LIN {X 0,Y 488.244,Z 843.404,A -85,B 0,C 180,E1 -6577.215,E2 -6577.215} C_VEL
LIN {X 0,Y 488.428,Z 836.225,A -85,B 0,C 180,E1 -6578.482,E2 -6578.482} C_VEL
LIN {X 0,Y 488.619,Z 827.431,A -85,B 0,C 180,E1 -6579.73,E2 -6579.73} C_VEL
LIN {X 0,Y 488.934,Z 817.433,A -85,B 0,C 180,E1 -6580.875,E2 -6580.875} C_VEL
LIN {X 0,Y 489.324,Z 806.303,A -85,B 0,C 180,E1 -6581.902,E2 -6581.902} C_VEL
LIN {X 0,Y 489.653,Z 795.065,A -85,B 0,C 180,E1 -6582.738,E2 -6582.738} C_VEL
LIN {X 0,Y 490.023,Z 782.384,A -85,B 0,C 180,E1 -6583.478,E2 -6583.478} C_VEL
LIN {X 0,Y 490.49,Z 769.48,A -85,B 0,C 180,E1 -6584.046,E2 -6584.046} C_VEL
LIN {X 0,Y 490.805,Z 756.071,A -85,B 0,C 180,E1 -6584.46,E2 -6584.46} C_VEL
LIN {X 0,Y 491.062,Z 737.319,A -85,B 0,C 180,E1 -6584.796,E2 -6584.796} C_VEL
LIN {X 0,Y 491.554,Z 664.239,A -85,B 0,C 180,E1 -6585.948,E2 -6585.948} C_VEL
LIN {X 0,Y 490.064,Z 652.447,A -85,B 0,C 180,E1 -6586.19,E2 -6586.19} C_VEL
LIN {X 0,Y 489.098,Z 638.268,A -85,B 0,C 180,E1 -6586.485,E2 -6586.485} C_VEL
LIN {X 0,Y 489.362,Z 617.504,A -85,B 0,C 180,E1 -6589.506,E2 -6589.506} C_VEL
LIN {X 0,Y 489.557,Z 597.975,A -85,B 0,C 180,E1 -6592.361,E2 -6592.361} C_VEL
LIN {X 0,Y 489.714,Z 578.159,A -85,B 0,C 180,E1 -6595.293,E2 -6595.293} C_VEL
LIN {X 0,Y 489.897,Z 557.152,A -85,B 0,C 180,E1 -6598.468,E2 -6598.468} C_VEL
LIN {X 0,Y 489.78,Z 545.178,A -85,B 0,C 180,E1 -6600.327,E2 -6600.327} C_VEL
LIN {X 0,Y 488.831,Z 539.598,A -85,B 0,C 180,E1 -6601.261,E2 -6601.261} C_VEL
LIN {X 0,Y 488.737,Z 539.605,A -85,B 0,C 180,E1 -6604.113,E2 -6604.113} C_VEL
LIN {X 0,Y 488.684,Z 539.613,A -85,B 0,C 180,E1 -6607.159,E2 -6607.159} C_VEL
LIN {X 0,Y 488.723,Z 539.606,A -85,B 0,C 180,E1 -6610.345,E2 -6610.345} C_VEL
LIN {X 0,Y 488.691,Z 539.608,A -85,B 0,C 180,E1 -6613.654,E2 -6613.654} C_VEL
LIN {X 0,Y 488.692,Z 539.611,A -85,B 0,C 180,E1 -6616.346,E2 -6616.346} C_VEL
LIN {X 0,Y 488.737,Z 539.602,A -85,B 0,C 180,E1 -6619.677,E2 -6619.677} C_VEL
LIN {X 0,Y 488.684,Z 539.615,A -85,B 0,C 180,E1 -6622.841,E2 -6622.841} C_VEL
LIN {X 0,Y 488.735,Z 539.604,A -85,B 0,C 180,E1 -6625.887,E2 -6625.887} C_VEL
LIN {X 0,Y 488.697,Z 539.612,A -85,B 0,C 180,E1 -6628.82,E2 -6628.82} C_VEL
LIN {X 0,Y 488.75,Z 539.602,A -85,B 0,C 180,E1 -6631.671,E2 -6631.671} C_VEL
LIN {X 0,Y 488.752,Z 539.608,A -85,B 0,C 180,E1 -6634.444,E2 -6634.444} C_VEL
LIN {X 0,Y 488.728,Z 539.607,A -85,B 0,C 180,E1 -6637.153,E2 -6637.153} C_VEL
LIN {X 0,Y 488.73,Z 539.607,A -85,B 0,C 180,E1 -6639.81,E2 -6639.81} C_VEL
LIN {X 0,Y 488.751,Z 539.609,A -85,B 0,C 180,E1 -6642.591,E2 -6642.591} C_VEL
LIN {X 0,Y 492.762,Z 551.195,A -85,B 0,C 180,E1 -6642.917,E2 -6642.917} C_VEL
LIN {X 0,Y 492.751,Z 584.57,A -85,B 0,C 180,E1 -6643.426,E2 -6643.426} C_VEL
LIN {X 0,Y 492.704,Z 599.838,A -85,B 0,C 180,E1 -6643.83,E2 -6643.83} C_VEL
LIN {X 0,Y 492.57,Z 614.087,A -85,B 0,C 180,E1 -6644.377,E2 -6644.377} C_VEL
LIN {X 0,Y 492.273,Z 626.69,A -85,B 0,C 180,E1 -6645.003,E2 -6645.003} C_VEL
LIN {X 0,Y 491.859,Z 639.98,A -85,B 0,C 180,E1 -6645.836,E2 -6645.836} C_VEL
LIN {X 0,Y 491.447,Z 653.278,A -85,B 0,C 180,E1 -6646.878,E2 -6646.878} C_VEL
LIN {X 0,Y 491.009,Z 664.22,A -85,B 0,C 180,E1 -6647.916,E2 -6647.916} C_VEL
LIN {X 0,Y 490.483,Z 674.33,A -85,B 0,C 180,E1 -6649.055,E2 -6649.055} C_VEL
LIN {X 0,Y 489.999,Z 683.621,A -85,B 0,C 180,E1 -6650.297,E2 -6650.297} C_VEL
LIN {X 0,Y 489.615,Z 692.638,A -85,B 0,C 180,E1 -6651.747,E2 -6651.747} C_VEL
LIN {X 0,Y 489.34,Z 699.094,A -85,B 0,C 180,E1 -6652.988,E2 -6652.988} C_VEL
LIN {X 0,Y 488.977,Z 704.583,A -85,B 0,C 180,E1 -6654.225,E2 -6654.225} C_VEL
LIN {X 0,Y 488.744,Z 710.483,A -85,B 0,C 180,E1 -6655.877,E2 -6655.877} C_VEL
LIN {X 0,Y 488.548,Z 714.977,A -85,B 0,C 180,E1 -6657.526,E2 -6657.526} C_VEL
LIN {X 0,Y 488.433,Z 718.193,A -85,B 0,C 180,E1 -6659.175,E2 -6659.175} C_VEL
LIN {X 0,Y 488.414,Z 720.216,A -85,B 0,C 180,E1 -6660.824,E2 -6660.824} C_VEL
LIN {X 0,Y 488.451,Z 721.099,A -85,B 0,C 180,E1 -6662.474,E2 -6662.474} C_VEL
LIN {X 0,Y 488.351,Z 720.88,A -85,B 0,C 180,E1 -6664.126,E2 -6664.126} C_VEL
LIN {X 0,Y 488.426,Z 719.509,A -85,B 0,C 180,E1 -6665.78,E2 -6665.78} C_VEL
LIN {X 0,Y 488.492,Z 716.945,A -85,B 0,C 180,E1 -6667.439,E2 -6667.439} C_VEL
LIN {X 0,Y 488.66,Z 713.137,A -85,B 0,C 180,E1 -6669.102,E2 -6669.102} C_VEL
LIN {X 0,Y 488.734,Z 708.023,A -85,B 0,C 180,E1 -6670.774,E2 -6670.774} C_VEL
LIN {X 0,Y 489.054,Z 701.415,A -85,B 0,C 180,E1 -6672.448,E2 -6672.448} C_VEL
LIN {X 0,Y 489.458,Z 693.105,A -85,B 0,C 180,E1 -6674.128,E2 -6674.128} C_VEL
LIN {X 0,Y 489.883,Z 684.147,A -85,B 0,C 180,E1 -6675.604,E2 -6675.604} C_VEL
LIN {X 0,Y 490.418,Z 673.246,A -85,B 0,C 180,E1 -6677.084,E2 -6677.084} C_VEL
LIN {X 0,Y 490.971,Z 661.901,A -85,B 0,C 180,E1 -6678.355,E2 -6678.355} C_VEL
LIN {X 0,Y 491.484,Z 650.595,A -85,B 0,C 180,E1 -6679.418,E2 -6679.418} C_VEL
LIN {X 0,Y 491.957,Z 638.327,A -85,B 0,C 180,E1 -6680.378,E2 -6680.378} C_VEL
LIN {X 0,Y 492.432,Z 624.976,A -85,B 0,C 180,E1 -6681.232,E2 -6681.232} C_VEL
LIN {X 0,Y 492.849,Z 612.015,A -85,B 0,C 180,E1 -6681.893,E2 -6681.893} C_VEL
LIN {X 0,Y 493.158,Z 597.332,A -85,B 0,C 180,E1 -6682.474,E2 -6682.474} C_VEL
LIN {X 0,Y 493.277,Z 584.102,A -85,B 0,C 180,E1 -6682.855,E2 -6682.855} C_VEL
LIN {X 0,Y 493.378,Z 564.328,A -85,B 0,C 180,E1 -6683.214,E2 -6683.214} C_VEL
LIN {X 0,Y 493.335,Z 552.237,A -85,B 0,C 180,E1 -6683.406,E2 -6683.406} C_VEL
LIN {X 0,Y 488.739,Z 539.609,A -85,B 0,C 180,E1 -6683.799,E2 -6683.799} C_VEL
LIN {X 0,Y 488.794,Z 539.595,A -85,B 0,C 180,E1 -6686.943,E2 -6686.943} C_VEL
LIN {X 0,Y 488.711,Z 539.608,A -85,B 0,C 180,E1 -6690.362,E2 -6690.362} C_VEL
LIN {X 0,Y 488.735,Z 539.602,A -85,B 0,C 180,E1 -6693.484,E2 -6693.484} C_VEL
LIN {X 0,Y 488.683,Z 539.613,A -85,B 0,C 180,E1 -6696.354,E2 -6696.354} C_VEL
LIN {X 0,Y 488.703,Z 539.604,A -85,B 0,C 180,E1 -6699.254,E2 -6699.254} C_VEL
LIN {X 0,Y 488.709,Z 539.605,A -85,B 0,C 180,E1 -6701.599,E2 -6701.599} C_VEL
LIN {X 0,Y 488.701,Z 539.607,A -85,B 0,C 180,E1 -6704.802,E2 -6704.802} C_VEL
LIN {X 0,Y 488.692,Z 539.606,A -85,B 0,C 180,E1 -6707.474,E2 -6707.474} C_VEL
LIN {X 0,Y 488.733,Z 539.601,A -85,B 0,C 180,E1 -6709.676,E2 -6709.676} C_VEL
LIN {X 0,Y 488.68,Z 539.611,A -85,B 0,C 180,E1 -6712.841,E2 -6712.841} C_VEL
LIN {X 0,Y 488.72,Z 539.606,A -85,B 0,C 180,E1 -6714.907,E2 -6714.907} C_VEL
LIN {X 0,Y 488.072,Z 539.684,A -85,B 0,C 180,E1 -6715.595,E2 -6715.595} C_VEL
LIN {X 0,Y 485.214,Z 540.046,A -85,B 0,C 180,E1 -6716.713,E2 -6716.713} C_VEL
LIN {X 0,Y 482.778,Z 540.35,A -85,B 0,C 180,E1 -6717.613,E2 -6717.613} C_VEL
LIN {X 0,Y 481.723,Z 540.479,A -85,B 0,C 180,E1 -6718.309,E2 -6718.309} C_VEL
LIN {X 0,Y 481.633,Z 540.488,A -85,B 0,C 180,E1 -6718.544,E2 -6718.544} C_VEL
LIN {X 0,Y 481.699,Z 540.478,A -85,B 0,C 180,E1 -6721.218,E2 -6721.218} C_VEL
LIN {X 0,Y 481.7,Z 540.478,A -85,B 0,C 180,E1 -6724.042,E2 -6724.042} C_VEL
LIN {X 0,Y 481.674,Z 540.488,A -85,B 0,C 180,E1 -6726.811,E2 -6726.811} C_VEL
LIN {X 0,Y 481.696,Z 540.478,A -85,B 0,C 180,E1 -6729.502,E2 -6729.502} C_VEL
LIN {X 0,Y 481.706,Z 540.477,A -85,B 0,C 180,E1 -6732.158,E2 -6732.158} C_VEL
LIN {X 0,Y 481.741,Z 540.48,A -85,B 0,C 180,E1 -6734.775,E2 -6734.775} C_VEL
LIN {X 0,Y 481.75,Z 540.471,A -85,B 0,C 180,E1 -6738.215,E2 -6738.215} C_VEL
LIN {X 0,Y 481.762,Z 540.471,A -85,B 0,C 180,E1 -6741.611,E2 -6741.611} C_VEL
LIN {X 0,Y 481.815,Z 540.463,A -85,B 0,C 180,E1 -6744.139,E2 -6744.139} C_VEL
LIN {X 0,Y 481.927,Z 540.452,A -85,B 0,C 180,E1 -6747.492,E2 -6747.492} C_VEL
LIN {X 0,Y 481.904,Z 540.456,A -85,B 0,C 180,E1 -6750.835,E2 -6750.835} C_VEL
LIN {X 0,Y 481.927,Z 540.45,A -85,B 0,C 180,E1 -6752.507,E2 -6752.507} C_VEL
LIN {X 0,Y 481.806,Z 540.465,A -85,B 0,C 180,E1 -6755.86,E2 -6755.86} C_VEL
LIN {X 0,Y 481.76,Z 540.469,A -85,B 0,C 180,E1 -6758.388,E2 -6758.388} C_VEL
LIN {X 0,Y 481.792,Z 540.469,A -85,B 0,C 180,E1 -6761.783,E2 -6761.783} C_VEL
LIN {X 0,Y 481.739,Z 540.478,A -85,B 0,C 180,E1 -6765.224,E2 -6765.224} C_VEL
LIN {X 0,Y 481.709,Z 540.476,A -85,B 0,C 180,E1 -6768.721,E2 -6768.721} C_VEL
LIN {X 0,Y 481.644,Z 540.491,A -85,B 0,C 180,E1 -6771.394,E2 -6771.394} C_VEL
LIN {X 0,Y 481.674,Z 540.482,A -85,B 0,C 180,E1 -6774.113,E2 -6774.113} C_VEL
LIN {X 0,Y 481.748,Z 540.473,A -85,B 0,C 180,E1 -6777.14,E2 -6777.14} C_VEL
LIN {X 0,Y 481.684,Z 540.487,A -85,B 0,C 180,E1 -6779.74,E2 -6779.74} C_VEL
LIN {X 0,Y 481.669,Z 540.481,A -85,B 0,C 180,E1 -6782.674,E2 -6782.674} C_VEL
LIN {X 0,Y 481.639,Z 540.492,A -85,B 0,C 180,E1 -6785.709,E2 -6785.709} C_VEL
LIN {X 0,Y 481.709,Z 540.478,A -85,B 0,C 180,E1 -6789.354,E2 -6789.354} C_VEL
LIN {X 0,Y 481.643,Z 540.489,A -85,B 0,C 180,E1 -6792.16,E2 -6792.16} C_VEL
LIN {X 0,Y 481.655,Z 540.486,A -85,B 0,C 180,E1 -6795.543,E2 -6795.543} C_VEL
LIN {X 0,Y 481.669,Z 540.489,A -85,B 0,C 180,E1 -6798.084,E2 -6798.084} C_VEL
LIN {X 0,Y 481.698,Z 540.477,A -85,B 0,C 180,E1 -6801.144,E2 -6801.144} C_VEL
LIN {X 0,Y 481.664,Z 540.483,A -85,B 0,C 180,E1 -6804.794,E2 -6804.794} C_VEL
LIN {X 0,Y 481.668,Z 540.482,A -85,B 0,C 180,E1 -6807.326,E2 -6807.326} C_VEL
LIN {X 0,Y 481.683,Z 540.487,A -85,B 0,C 180,E1 -6808.46,E2 -6808.46} C_VEL
LIN {X 0,Y 485.781,Z 552.58,A -85,B 0,C 180,E1 -6808.819,E2 -6808.819} C_VEL
LIN {X 0,Y 485.413,Z 598.433,A -85,B 0,C 180,E1 -6809.553,E2 -6809.553} C_VEL
LIN {X 0,Y 485.199,Z 612.867,A -85,B 0,C 180,E1 -6809.951,E2 -6809.951} C_VEL
LIN {X 0,Y 484.98,Z 626.879,A -85,B 0,C 180,E1 -6810.52,E2 -6810.52} C_VEL
LIN {X 0,Y 484.584,Z 639.004,A -85,B 0,C 180,E1 -6811.169,E2 -6811.169} C_VEL
LIN {X 0,Y 484.144,Z 650.859,A -85,B 0,C 180,E1 -6811.968,E2 -6811.968} C_VEL
LIN {X 0,Y 483.677,Z 663.087,A -85,B 0,C 180,E1 -6812.995,E2 -6812.995} C_VEL
LIN {X 0,Y 483.146,Z 674.101,A -85,B 0,C 180,E1 -6814.127,E2 -6814.127} C_VEL
LIN {X 0,Y 482.709,Z 683.193,A -85,B 0,C 180,E1 -6815.255,E2 -6815.255} C_VEL
LIN {X 0,Y 482.308,Z 692.392,A -85,B 0,C 180,E1 -6816.635,E2 -6816.635} C_VEL
LIN {X 0,Y 481.953,Z 700.64,A -85,B 0,C 180,E1 -6818.171,E2 -6818.171} C_VEL
LIN {X 0,Y 481.662,Z 706.428,A -85,B 0,C 180,E1 -6819.502,E2 -6819.502} C_VEL
LIN {X 0,Y 481.525,Z 711.062,A -85,B 0,C 180,E1 -6820.829,E2 -6820.829} C_VEL
LIN {X 0,Y 481.381,Z 714.67,A -85,B 0,C 180,E1 -6822.146,E2 -6822.146} C_VEL
LIN {X 0,Y 481.227,Z 718.115,A -85,B 0,C 180,E1 -6823.89,E2 -6823.89} C_VEL
LIN {X 0,Y 481.178,Z 720.03,A -85,B 0,C 180,E1 -6825.624,E2 -6825.624} C_VEL
LIN {X 0,Y 481.21,Z 720.536,A -85,B 0,C 180,E1 -6827.346,E2 -6827.346} C_VEL
LIN {X 0,Y 481.237,Z 719.683,A -85,B 0,C 180,E1 -6829.056,E2 -6829.056} C_VEL
LIN {X 0,Y 481.306,Z 717.471,A -85,B 0,C 180,E1 -6830.757,E2 -6830.757} C_VEL
LIN {X 0,Y 481.496,Z 713.828,A -85,B 0,C 180,E1 -6832.452,E2 -6832.452} C_VEL
LIN {X 0,Y 481.709,Z 708.629,A -85,B 0,C 180,E1 -6834.139,E2 -6834.139} C_VEL
LIN {X 0,Y 481.874,Z 703.677,A -85,B 0,C 180,E1 -6835.399,E2 -6835.399} C_VEL
LIN {X 0,Y 482.231,Z 696.478,A -85,B 0,C 180,E1 -6836.867,E2 -6836.867} C_VEL
LIN {X 0,Y 482.631,Z 687.563,A -85,B 0,C 180,E1 -6838.331,E2 -6838.331} C_VEL
LIN {X 0,Y 483.138,Z 678.174,A -85,B 0,C 180,E1 -6839.584,E2 -6839.584} C_VEL
LIN {X 0,Y 483.541,Z 667.763,A -85,B 0,C 180,E1 -6840.729,E2 -6840.729} C_VEL
LIN {X 0,Y 484.075,Z 656.066,A -85,B 0,C 180,E1 -6841.768,E2 -6841.768} C_VEL
LIN {X 0,Y 484.511,Z 644.559,A -85,B 0,C 180,E1 -6842.598,E2 -6842.598} C_VEL
LIN {X 0,Y 484.855,Z 631.922,A -85,B 0,C 180,E1 -6843.324,E2 -6843.324} C_VEL
LIN {X 0,Y 485.123,Z 618.257,A -85,B 0,C 180,E1 -6843.92,E2 -6843.92} C_VEL
LIN {X 0,Y 485.253,Z 604.829,A -85,B 0,C 180,E1 -6844.335,E2 -6844.335} C_VEL
LIN {X 0,Y 485.288,Z 589.639,A -85,B 0,C 180,E1 -6844.621,E2 -6844.621} C_VEL
LIN {X 0,Y 485.423,Z 551.252,A -85,B 0,C 180,E1 -6845.205,E2 -6845.205} C_VEL
LIN {X 0,Y 481.805,Z 540.474,A -85,B 0,C 180,E1 -6845.52,E2 -6845.52} C_VEL
LIN {X 0,Y 481.824,Z 540.47,A -85,B 0,C 180,E1 -6847.544,E2 -6847.544} C_VEL
LIN {X 0,Y 481.713,Z 540.48,A -85,B 0,C 180,E1 -6850.934,E2 -6850.934} C_VEL
LIN {X 0,Y 481.692,Z 540.488,A -85,B 0,C 180,E1 -6853.5,E2 -6853.5} C_VEL
LIN {X 0,Y 481.694,Z 540.483,A -85,B 0,C 180,E1 -6856.094,E2 -6856.094} C_VEL
LIN {X 0,Y 481.709,Z 540.48,A -85,B 0,C 180,E1 -6858.722,E2 -6858.722} C_VEL
LIN {X 0,Y 481.644,Z 540.492,A -85,B 0,C 180,E1 -6861.395,E2 -6861.395} C_VEL
LIN {X 0,Y 481.675,Z 540.483,A -85,B 0,C 180,E1 -6864.114,E2 -6864.114} C_VEL
LIN {X 0,Y 481.75,Z 540.476,A -85,B 0,C 180,E1 -6867.141,E2 -6867.141} C_VEL
LIN {X 0,Y 481.686,Z 540.48,A -85,B 0,C 180,E1 -6869.741,E2 -6869.741} C_VEL
LIN {X 0,Y 481.671,Z 540.478,A -85,B 0,C 180,E1 -6872.675,E2 -6872.675} C_VEL
LIN {X 0,Y 481.636,Z 540.487,A -85,B 0,C 180,E1 -6875.71,E2 -6875.71} C_VEL
LIN {X 0,Y 481.67,Z 540.484,A -85,B 0,C 180,E1 -6878.86,E2 -6878.86} C_VEL
LIN {X 0,Y 481.661,Z 540.483,A -85,B 0,C 180,E1 -6881.915,E2 -6881.915} C_VEL
LIN {X 0,Y 481.659,Z 540.484,A -85,B 0,C 180,E1 -6884.458,E2 -6884.458} C_VEL
LIN {X 0,Y 481.647,Z 540.485,A -85,B 0,C 180,E1 -6887.84,E2 -6887.84} C_VEL
LIN {X 0,Y 481.68,Z 540.484,A -85,B 0,C 180,E1 -6890.652,E2 -6890.652} C_VEL
LIN {X 0,Y 481.631,Z 540.495,A -85,B 0,C 180,E1 -6893.376,E2 -6893.376} C_VEL
LIN {X 0,Y 481.731,Z 540.556,A -85,B 0,C 180,E1 -6895.811,E2 -6895.811} C_VEL
LIN {X 0,Y 485.054,Z 555.824,A -85,B 0,C 180,E1 -6898.745,E2 -6898.745} C_VEL
LIN {X 0,Y 484.971,Z 563.014,A -85,B 0,C 180,E1 -6900.004,E2 -6900.004} C_VEL
LIN {X 0,Y 484.154,Z 580.75,A -85,B 0,C 180,E1 -6903.024,E2 -6903.024} C_VEL
LIN {X 0,Y 483.441,Z 599.885,A -85,B 0,C 180,E1 -6906.214,E2 -6906.214} C_VEL
LIN {X 0,Y 482.823,Z 618.961,A -85,B 0,C 180,E1 -6909.331,E2 -6909.331} C_VEL
LIN {X 0,Y 482.197,Z 639.335,A -85,B 0,C 180,E1 -6912.616,E2 -6912.616} C_VEL
LIN {X 0,Y 482.116,Z 643.051,A -85,B 0,C 180,E1 -6913.18,E2 -6913.18} C_VEL
LIN {X 0,Y 485.175,Z 666.865,A -85,B 0,C 180,E1 -6913.723,E2 -6913.723} C_VEL
LIN {X 0,Y 484.568,Z 728.928,A -85,B 0,C 180,E1 -6914.733,E2 -6914.733} C_VEL
LIN {X 0,Y 484.207,Z 755.366,A -85,B 0,C 180,E1 -6915.205,E2 -6915.205} C_VEL
LIN {X 0,Y 483.804,Z 768.384,A -85,B 0,C 180,E1 -6915.596,E2 -6915.596} C_VEL
LIN {X 0,Y 483.31,Z 781.583,A -85,B 0,C 180,E1 -6916.172,E2 -6916.172} C_VEL
LIN {X 0,Y 482.855,Z 793.278,A -85,B 0,C 180,E1 -6916.855,E2 -6916.855} C_VEL
LIN {X 0,Y 482.513,Z 804.426,A -85,B 0,C 180,E1 -6917.681,E2 -6917.681} C_VEL
LIN {X 0,Y 482.035,Z 815.029,A -85,B 0,C 180,E1 -6918.649,E2 -6918.649} C_VEL
LIN {X 0,Y 481.654,Z 824.401,A -85,B 0,C 180,E1 -6919.704,E2 -6919.704} C_VEL
LIN {X 0,Y 481.385,Z 833.559,A -85,B 0,C 180,E1 -6920.971,E2 -6920.971} C_VEL
LIN {X 0,Y 481.19,Z 840.958,A -85,B 0,C 180,E1 -6922.236,E2 -6922.236} C_VEL
LIN {X 0,Y 481.088,Z 847.616,A -85,B 0,C 180,E1 -6923.685,E2 -6923.685} C_VEL
LIN {X 0,Y 481.004,Z 852.178,A -85,B 0,C 180,E1 -6924.971,E2 -6924.971} C_VEL
LIN {X 0,Y 481.036,Z 854.544,A -85,B 0,C 180,E1 -6925.811,E2 -6925.811} C_VEL
LIN {X 0,Y 481.018,Z 856.455,A -85,B 0,C 180,E1 -6926.65,E2 -6926.65} C_VEL
LIN {X 0,Y 481.004,Z 857.885,A -85,B 0,C 180,E1 -6927.488,E2 -6927.488} C_VEL
LIN {X 0,Y 480.963,Z 858.886,A -85,B 0,C 180,E1 -6928.326,E2 -6928.326} C_VEL
LIN {X 0,Y 481.035,Z 859.663,A -85,B 0,C 180,E1 -6930,E2 -6930} C_VEL
LIN {X 0,Y 480.984,Z 858.715,A -85,B 0,C 180,E1 -6931.675,E2 -6931.675} C_VEL
LIN {X 0,Y 481.036,Z 857.614,A -85,B 0,C 180,E1 -6932.513,E2 -6932.513} C_VEL
LIN {X 0,Y 481.051,Z 856.087,A -85,B 0,C 180,E1 -6933.351,E2 -6933.351} C_VEL
LIN {X 0,Y 481.067,Z 852.918,A -85,B 0,C 180,E1 -6934.609,E2 -6934.609} C_VEL
LIN {X 0,Y 481.156,Z 847.635,A -85,B 0,C 180,E1 -6936.128,E2 -6936.128} C_VEL
LIN {X 0,Y 481.237,Z 841.023,A -85,B 0,C 180,E1 -6937.553,E2 -6937.553} C_VEL
LIN {X 0,Y 481.368,Z 833.636,A -85,B 0,C 180,E1 -6938.819,E2 -6938.819} C_VEL
LIN {X 0,Y 481.607,Z 824.427,A -85,B 0,C 180,E1 -6940.086,E2 -6940.086} C_VEL
LIN {X 0,Y 481.946,Z 813.957,A -85,B 0,C 180,E1 -6941.248,E2 -6941.248} C_VEL
LIN {X 0,Y 482.262,Z 804.328,A -85,B 0,C 180,E1 -6942.122,E2 -6942.122} C_VEL
LIN {X 0,Y 482.706,Z 793.375,A -85,B 0,C 180,E1 -6942.936,E2 -6942.936} C_VEL
LIN {X 0,Y 483.088,Z 780.772,A -85,B 0,C 180,E1 -6943.675,E2 -6943.675} C_VEL
LIN {X 0,Y 483.528,Z 767.798,A -85,B 0,C 180,E1 -6944.252,E2 -6944.252} C_VEL
LIN {X 0,Y 483.909,Z 754.321,A -85,B 0,C 180,E1 -6944.67,E2 -6944.67} C_VEL
LIN {X 0,Y 484.171,Z 735.562,A -85,B 0,C 180,E1 -6945.012,E2 -6945.012} C_VEL
LIN {X 0,Y 484.673,Z 664.75,A -85,B 0,C 180,E1 -6946.162,E2 -6946.162} C_VEL
LIN {X 0,Y 483.259,Z 653.156,A -85,B 0,C 180,E1 -6946.413,E2 -6946.413} C_VEL
LIN {X 0,Y 482.039,Z 636.017,A -85,B 0,C 180,E1 -6946.759,E2 -6946.759} C_VEL
LIN {X 0,Y 482.289,Z 615.418,A -85,B 0,C 180,E1 -6949.804,E2 -6949.804} C_VEL
LIN {X 0,Y 482.498,Z 595.939,A -85,B 0,C 180,E1 -6952.706,E2 -6952.706} C_VEL
LIN {X 0,Y 482.692,Z 574.794,A -85,B 0,C 180,E1 -6955.9,E2 -6955.9} C_VEL
LIN {X 0,Y 482.862,Z 555.22,A -85,B 0,C 180,E1 -6958.929,E2 -6958.929} C_VEL
LIN {X 0,Y 482.7,Z 545.998,A -85,B 0,C 180,E1 -6960.395,E2 -6960.395} C_VEL
LIN {X 0,Y 481.764,Z 540.478,A -85,B 0,C 180,E1 -6961.343,E2 -6961.343} C_VEL
LIN {X 0,Y 481.695,Z 540.486,A -85,B 0,C 180,E1 -6964.682,E2 -6964.682} C_VEL
LIN {X 0,Y 481.659,Z 540.484,A -85,B 0,C 180,E1 -6968.007,E2 -6968.007} C_VEL
LIN {X 0,Y 481.66,Z 540.489,A -85,B 0,C 180,E1 -6971.042,E2 -6971.042} C_VEL
LIN {X 0,Y 481.664,Z 540.487,A -85,B 0,C 180,E1 -6974.457,E2 -6974.457} C_VEL
LIN {X 0,Y 481.653,Z 540.485,A -85,B 0,C 180,E1 -6977.839,E2 -6977.839} C_VEL
LIN {X 0,Y 481.685,Z 540.485,A -85,B 0,C 180,E1 -6980.651,E2 -6980.651} C_VEL
LIN {X 0,Y 481.632,Z 540.489,A -85,B 0,C 180,E1 -6983.376,E2 -6983.376} C_VEL
LIN {X 0,Y 481.714,Z 540.482,A -85,B 0,C 180,E1 -6986.33,E2 -6986.33} C_VEL
LIN {X 0,Y 481.655,Z 540.485,A -85,B 0,C 180,E1 -6989.417,E2 -6989.417} C_VEL
LIN {X 0,Y 481.705,Z 540.484,A -85,B 0,C 180,E1 -6992.168,E2 -6992.168} C_VEL
LIN {X 0,Y 481.723,Z 540.481,A -85,B 0,C 180,E1 -6994.97,E2 -6994.97} C_VEL
LIN {X 0,Y 481.654,Z 540.489,A -85,B 0,C 180,E1 -6997.705,E2 -6997.705} C_VEL
LIN {X 0,Y 481.71,Z 540.485,A -85,B 0,C 180,E1 -7000.393,E2 -7000.393} C_VEL
LIN {X 0,Y 481.704,Z 540.487,A -85,B 0,C 180,E1 -7002.33,E2 -7002.33} C_VEL
LIN {X 0,Y 486.013,Z 552.722,A -85,B 0,C 180,E1 -7002.687,E2 -7002.687} C_VEL
LIN {X 0,Y 485.966,Z 586.169,A -85,B 0,C 180,E1 -7003.207,E2 -7003.207} C_VEL
LIN {X 0,Y 485.923,Z 601.32,A -85,B 0,C 180,E1 -7003.617,E2 -7003.617} C_VEL
LIN {X 0,Y 485.81,Z 615.185,A -85,B 0,C 180,E1 -7004.153,E2 -7004.153} C_VEL
LIN {X 0,Y 485.522,Z 627.851,A -85,B 0,C 180,E1 -7004.789,E2 -7004.789} C_VEL
LIN {X 0,Y 485.077,Z 641.2,A -85,B 0,C 180,E1 -7005.634,E2 -7005.634} C_VEL
LIN {X 0,Y 484.638,Z 654.535,A -85,B 0,C 180,E1 -7006.69,E2 -7006.69} C_VEL
LIN {X 0,Y 484.18,Z 665.492,A -85,B 0,C 180,E1 -7007.743,E2 -7007.743} C_VEL
LIN {X 0,Y 483.638,Z 675.579,A -85,B 0,C 180,E1 -7008.898,E2 -7008.898} C_VEL
LIN {X 0,Y 483.107,Z 684.844,A -85,B 0,C 180,E1 -7010.158,E2 -7010.158} C_VEL
LIN {X 0,Y 482.704,Z 693.827,A -85,B 0,C 180,E1 -7011.628,E2 -7011.628} C_VEL
LIN {X 0,Y 482.393,Z 700.275,A -85,B 0,C 180,E1 -7012.886,E2 -7012.886} C_VEL
LIN {X 0,Y 482.012,Z 705.761,A -85,B 0,C 180,E1 -7014.142,E2 -7014.142} C_VEL
LIN {X 0,Y 481.759,Z 711.647,A -85,B 0,C 180,E1 -7015.817,E2 -7015.817} C_VEL
LIN {X 0,Y 481.567,Z 716.116,A -85,B 0,C 180,E1 -7017.49,E2 -7017.49} C_VEL
LIN {X 0,Y 481.423,Z 719.307,A -85,B 0,C 180,E1 -7019.163,E2 -7019.163} C_VEL
LIN {X 0,Y 481.403,Z 721.298,A -85,B 0,C 180,E1 -7020.836,E2 -7020.836} C_VEL
LIN {X 0,Y 481.438,Z 722.139,A -85,B 0,C 180,E1 -7022.51,E2 -7022.51} C_VEL
LIN {X 0,Y 481.328,Z 721.872,A -85,B 0,C 180,E1 -7024.186,E2 -7024.186} C_VEL
LIN {X 0,Y 481.419,Z 720.443,A -85,B 0,C 180,E1 -7025.865,E2 -7025.865} C_VEL
LIN {X 0,Y 481.48,Z 717.837,A -85,B 0,C 180,E1 -7027.548,E2 -7027.548} C_VEL
LIN {X 0,Y 481.661,Z 713.962,A -85,B 0,C 180,E1 -7029.236,E2 -7029.236} C_VEL
LIN {X 0,Y 481.769,Z 708.768,A -85,B 0,C 180,E1 -7030.932,E2 -7030.932} C_VEL
LIN {X 0,Y 482.097,Z 702.072,A -85,B 0,C 180,E1 -7032.631,E2 -7032.631} C_VEL
LIN {X 0,Y 482.489,Z 694.778,A -85,B 0,C 180,E1 -7034.121,E2 -7034.121} C_VEL
LIN {X 0,Y 482.93,Z 685.947,A -85,B 0,C 180,E1 -7035.618,E2 -7035.618} C_VEL
LIN {X 0,Y 483.409,Z 676.866,A -85,B 0,C 180,E1 -7036.904,E2 -7036.904} C_VEL
LIN {X 0,Y 483.943,Z 666.047,A -85,B 0,C 180,E1 -7038.193,E2 -7038.193} C_VEL
LIN {X 0,Y 484.508,Z 654.799,A -85,B 0,C 180,E1 -7039.315,E2 -7039.315} C_VEL
LIN {X 0,Y 485.005,Z 642.369,A -85,B 0,C 180,E1 -7040.351,E2 -7040.351} C_VEL
LIN {X 0,Y 485.491,Z 629.731,A -85,B 0,C 180,E1 -7041.217,E2 -7041.217} C_VEL
LIN {X 0,Y 485.967,Z 615.958,A -85,B 0,C 180,E1 -7041.975,E2 -7041.975} C_VEL
LIN {X 0,Y 486.365,Z 601.419,A -85,B 0,C 180,E1 -7042.591,E2 -7042.591} C_VEL
LIN {X 0,Y 486.473,Z 587.942,A -85,B 0,C 180,E1 -7043.02,E2 -7043.02} C_VEL
LIN {X 0,Y 486.608,Z 572.08,A -85,B 0,C 180,E1 -7043.345,E2 -7043.345} C_VEL
LIN {X 0,Y 486.585,Z 553.784,A -85,B 0,C 180,E1 -7043.641,E2 -7043.641} C_VEL
LIN {X 0,Y 481.684,Z 540.487,A -85,B 0,C 180,E1 -7044.062,E2 -7044.062} C_VEL
LIN {X 0,Y 481.749,Z 540.473,A -85,B 0,C 180,E1 -7047.139,E2 -7047.139} C_VEL
LIN {X 0,Y 481.68,Z 540.486,A -85,B 0,C 180,E1 -7049.741,E2 -7049.741} C_VEL
LIN {X 0,Y 481.673,Z 540.482,A -85,B 0,C 180,E1 -7052.674,E2 -7052.674} C_VEL
LIN {X 0,Y 481.637,Z 540.488,A -85,B 0,C 180,E1 -7055.709,E2 -7055.709} C_VEL
LIN {X 0,Y 481.672,Z 540.481,A -85,B 0,C 180,E1 -7058.858,E2 -7058.858} C_VEL
LIN {X 0,Y 481.654,Z 540.487,A -85,B 0,C 180,E1 -7061.912,E2 -7061.912} C_VEL
LIN {X 0,Y 481.655,Z 540.489,A -85,B 0,C 180,E1 -7064.457,E2 -7064.457} C_VEL
LIN {X 0,Y 481.648,Z 540.485,A -85,B 0,C 180,E1 -7067.839,E2 -7067.839} C_VEL
LIN {X 0,Y 481.68,Z 540.485,A -85,B 0,C 180,E1 -7070.651,E2 -7070.651} C_VEL
LIN {X 0,Y 481.628,Z 540.486,A -85,B 0,C 180,E1 -7073.375,E2 -7073.375} C_VEL
LIN {X 0,Y 481.709,Z 540.482,A -85,B 0,C 180,E1 -7076.33,E2 -7076.33} C_VEL
LIN {X 0,Y 481.633,Z 540.488,A -85,B 0,C 180,E1 -7078.544,E2 -7078.544} C_VEL
LIN {X 0,Y 480.954,Z 540.572,A -85,B 0,C 180,E1 -7079.243,E2 -7079.243} C_VEL
LIN {X 0,Y 478.104,Z 540.931,A -85,B 0,C 180,E1 -7080.377,E2 -7080.377} C_VEL
LIN {X 0,Y 475.721,Z 541.224,A -85,B 0,C 180,E1 -7081.292,E2 -7081.292} C_VEL
LIN {X 0,Y 474.725,Z 541.347,A -85,B 0,C 180,E1 -7081.998,E2 -7081.998} C_VEL
LIN {X 0,Y 474.659,Z 541.357,A -85,B 0,C 180,E1 -7082.237,E2 -7082.237} C_VEL
LIN {X 0,Y 474.658,Z 541.354,A -85,B 0,C 180,E1 -7085.507,E2 -7085.507} C_VEL
LIN {X 0,Y 474.67,Z 541.356,A -85,B 0,C 180,E1 -7089.185,E2 -7089.185} C_VEL
LIN {X 0,Y 474.656,Z 541.354,A -85,B 0,C 180,E1 -7091.884,E2 -7091.884} C_VEL
LIN {X 0,Y 474.699,Z 541.353,A -85,B 0,C 180,E1 -7094.544,E2 -7094.544} C_VEL
LIN {X 0,Y 474.703,Z 541.349,A -85,B 0,C 180,E1 -7098.037,E2 -7098.037} C_VEL
LIN {X 0,Y 474.727,Z 541.348,A -85,B 0,C 180,E1 -7101.486,E2 -7101.486} C_VEL
LIN {X 0,Y 474.777,Z 541.339,A -85,B 0,C 180,E1 -7104.052,E2 -7104.052} C_VEL
LIN {X 0,Y 474.893,Z 541.329,A -85,B 0,C 180,E1 -7107.455,E2 -7107.455} C_VEL
LIN {X 0,Y 474.91,Z 541.323,A -85,B 0,C 180,E1 -7109.999,E2 -7109.999} C_VEL
LIN {X 0,Y 474.893,Z 541.326,A -85,B 0,C 180,E1 -7112.544,E2 -7112.544} C_VEL
LIN {X 0,Y 474.769,Z 541.341,A -85,B 0,C 180,E1 -7115.947,E2 -7115.947} C_VEL
LIN {X 0,Y 474.725,Z 541.346,A -85,B 0,C 180,E1 -7118.513,E2 -7118.513} C_VEL
LIN {X 0,Y 474.736,Z 541.346,A -85,B 0,C 180,E1 -7121.961,E2 -7121.961} C_VEL
LIN {X 0,Y 474.677,Z 541.356,A -85,B 0,C 180,E1 -7125.768,E2 -7125.768} C_VEL
LIN {X 0,Y 474.662,Z 541.356,A -85,B 0,C 180,E1 -7129.01,E2 -7129.01} C_VEL
LIN {X 0,Y 474.588,Z 541.369,A -85,B 0,C 180,E1 -7131.728,E2 -7131.728} C_VEL
LIN {X 0,Y 474.656,Z 541.355,A -85,B 0,C 180,E1 -7134.492,E2 -7134.492} C_VEL
LIN {X 0,Y 474.695,Z 541.354,A -85,B 0,C 180,E1 -7137.338,E2 -7137.338} C_VEL
LIN {X 0,Y 474.606,Z 541.361,A -85,B 0,C 180,E1 -7140.811,E2 -7140.811} C_VEL
LIN {X 0,Y 474.634,Z 541.363,A -85,B 0,C 180,E1 -7143.984,E2 -7143.984} C_VEL
LIN {X 0,Y 474.571,Z 541.365,A -85,B 0,C 180,E1 -7146.9,E2 -7146.9} C_VEL
LIN {X 0,Y 474.646,Z 541.361,A -85,B 0,C 180,E1 -7149.651,E2 -7149.651} C_VEL
LIN {X 0,Y 474.61,Z 541.36,A -85,B 0,C 180,E1 -7152.934,E2 -7152.934} C_VEL
LIN {X 0,Y 474.613,Z 541.367,A -85,B 0,C 180,E1 -7155.896,E2 -7155.896} C_VEL
LIN {X 0,Y 474.641,Z 541.356,A -85,B 0,C 180,E1 -7159.038,E2 -7159.038} C_VEL
LIN {X 0,Y 474.615,Z 541.363,A -85,B 0,C 180,E1 -7161.702,E2 -7161.702} C_VEL
LIN {X 0,Y 474.626,Z 541.36,A -85,B 0,C 180,E1 -7164.726,E2 -7164.726} C_VEL
LIN {X 0,Y 474.619,Z 541.366,A -85,B 0,C 180,E1 -7168.011,E2 -7168.011} C_VEL
LIN {X 0,Y 474.635,Z 541.365,A -85,B 0,C 180,E1 -7168.206,E2 -7168.206} C_VEL
LIN {X 0,Y 478.999,Z 553.6,A -85,B 0,C 180,E1 -7168.587,E2 -7168.587} C_VEL
LIN {X 0,Y 478.56,Z 599.976,A -85,B 0,C 180,E1 -7169.345,E2 -7169.345} C_VEL
LIN {X 0,Y 478.392,Z 614.495,A -85,B 0,C 180,E1 -7169.761,E2 -7169.761} C_VEL
LIN {X 0,Y 478.129,Z 628.492,A -85,B 0,C 180,E1 -7170.346,E2 -7170.346} C_VEL
LIN {X 0,Y 477.679,Z 641.566,A -85,B 0,C 180,E1 -7171.074,E2 -7171.074} C_VEL
LIN {X 0,Y 477.241,Z 654.43,A -85,B 0,C 180,E1 -7171.99,E2 -7171.99} C_VEL
LIN {X 0,Y 476.699,Z 666.349,A -85,B 0,C 180,E1 -7173.042,E2 -7173.042} C_VEL
LIN {X 0,Y 476.179,Z 677.048,A -85,B 0,C 180,E1 -7174.197,E2 -7174.197} C_VEL
LIN {X 0,Y 475.667,Z 687.332,A -85,B 0,C 180,E1 -7175.563,E2 -7175.563} C_VEL
LIN {X 0,Y 475.256,Z 695.754,A -85,B 0,C 180,E1 -7176.929,E2 -7176.929} C_VEL
LIN {X 0,Y 474.925,Z 702.636,A -85,B 0,C 180,E1 -7178.288,E2 -7178.288} C_VEL
LIN {X 0,Y 474.657,Z 708.234,A -85,B 0,C 180,E1 -7179.638,E2 -7179.638} C_VEL
LIN {X 0,Y 474.494,Z 712.72,A -85,B 0,C 180,E1 -7180.983,E2 -7180.983} C_VEL
LIN {X 0,Y 474.29,Z 717.138,A -85,B 0,C 180,E1 -7182.761,E2 -7182.761} C_VEL
LIN {X 0,Y 474.177,Z 720.006,A -85,B 0,C 180,E1 -7184.527,E2 -7184.527} C_VEL
LIN {X 0,Y 474.181,Z 721.412,A -85,B 0,C 180,E1 -7186.283,E2 -7186.283} C_VEL
LIN {X 0,Y 474.249,Z 721.385,A -85,B 0,C 180,E1 -7188.026,E2 -7188.026} C_VEL
LIN {X 0,Y 474.261,Z 720.006,A -85,B 0,C 180,E1 -7189.757,E2 -7189.757} C_VEL
LIN {X 0,Y 474.346,Z 717.251,A -85,B 0,C 180,E1 -7191.48,E2 -7191.48} C_VEL
LIN {X 0,Y 474.639,Z 713.023,A -85,B 0,C 180,E1 -7193.197,E2 -7193.197} C_VEL
LIN {X 0,Y 474.781,Z 708.804,A -85,B 0,C 180,E1 -7194.479,E2 -7194.479} C_VEL
LIN {X 0,Y 474.984,Z 703.625,A -85,B 0,C 180,E1 -7195.758,E2 -7195.758} C_VEL
LIN {X 0,Y 475.347,Z 696.182,A -85,B 0,C 180,E1 -7197.246,E2 -7197.246} C_VEL
LIN {X 0,Y 475.764,Z 688.357,A -85,B 0,C 180,E1 -7198.519,E2 -7198.519} C_VEL
LIN {X 0,Y 476.268,Z 678.909,A -85,B 0,C 180,E1 -7199.789,E2 -7199.789} C_VEL
LIN {X 0,Y 476.721,Z 668.358,A -85,B 0,C 180,E1 -7200.951,E2 -7200.951} C_VEL
LIN {X 0,Y 477.26,Z 656.564,A -85,B 0,C 180,E1 -7202.005,E2 -7202.005} C_VEL
LIN {X 0,Y 477.727,Z 644.922,A -85,B 0,C 180,E1 -7202.846,E2 -7202.846} C_VEL
LIN {X 0,Y 478.09,Z 632.097,A -85,B 0,C 180,E1 -7203.582,E2 -7203.582} C_VEL
LIN {X 0,Y 478.356,Z 618.138,A -85,B 0,C 180,E1 -7204.187,E2 -7204.187} C_VEL
LIN {X 0,Y 478.448,Z 603.934,A -85,B 0,C 180,E1 -7204.608,E2 -7204.608} C_VEL
LIN {X 0,Y 478.57,Z 580.675,A -85,B 0,C 180,E1 -7205.003,E2 -7205.003} C_VEL
LIN {X 0,Y 478.647,Z 552.635,A -85,B 0,C 180,E1 -7205.439,E2 -7205.439} C_VEL
LIN {X 0,Y 474.78,Z 541.347,A -85,B 0,C 180,E1 -7205.788,E2 -7205.788} C_VEL
LIN {X 0,Y 474.725,Z 541.351,A -85,B 0,C 180,E1 -7208.514,E2 -7208.514} C_VEL
LIN {X 0,Y 474.736,Z 541.352,A -85,B 0,C 180,E1 -7211.962,E2 -7211.962} C_VEL
LIN {X 0,Y 474.677,Z 541.361,A -85,B 0,C 180,E1 -7215.768,E2 -7215.768} C_VEL
LIN {X 0,Y 474.662,Z 541.36,A -85,B 0,C 180,E1 -7219.011,E2 -7219.011} C_VEL
LIN {X 0,Y 474.588,Z 541.37,A -85,B 0,C 180,E1 -7221.729,E2 -7221.729} C_VEL
LIN {X 0,Y 474.657,Z 541.356,A -85,B 0,C 180,E1 -7224.493,E2 -7224.493} C_VEL
LIN {X 0,Y 474.696,Z 541.355,A -85,B 0,C 180,E1 -7227.339,E2 -7227.339} C_VEL
LIN {X 0,Y 474.608,Z 541.36,A -85,B 0,C 180,E1 -7230.812,E2 -7230.812} C_VEL
LIN {X 0,Y 474.635,Z 541.355,A -85,B 0,C 180,E1 -7233.984,E2 -7233.984} C_VEL
LIN {X 0,Y 474.571,Z 541.367,A -85,B 0,C 180,E1 -7236.9,E2 -7236.9} C_VEL
LIN {X 0,Y 474.626,Z 541.362,A -85,B 0,C 180,E1 -7239.648,E2 -7239.648} C_VEL
LIN {X 0,Y 474.634,Z 541.362,A -85,B 0,C 180,E1 -7242.933,E2 -7242.933} C_VEL
LIN {X 0,Y 474.608,Z 541.362,A -85,B 0,C 180,E1 -7245.896,E2 -7245.896} C_VEL
LIN {X 0,Y 474.627,Z 541.361,A -85,B 0,C 180,E1 -7249.041,E2 -7249.041} C_VEL
LIN {X 0,Y 474.61,Z 541.366,A -85,B 0,C 180,E1 -7251.705,E2 -7251.705} C_VEL
LIN {X 0,Y 474.655,Z 541.363,A -85,B 0,C 180,E1 -7255.247,E2 -7255.247} C_VEL
LIN {X 0,Y 474.67,Z 541.51,A -85,B 0,C 180,E1 -7255.57,E2 -7255.57} C_VEL
LIN {X 0,Y 477.796,Z 555.783,A -85,B 0,C 180,E1 -7258.36,E2 -7258.36} C_VEL
LIN {X 0,Y 478.268,Z 559.479,A -85,B 0,C 180,E1 -7259.049,E2 -7259.049} C_VEL
LIN {X 0,Y 477.433,Z 577.237,A -85,B 0,C 180,E1 -7262.141,E2 -7262.141} C_VEL
LIN {X 0,Y 476.585,Z 596.261,A -85,B 0,C 180,E1 -7265.381,E2 -7265.381} C_VEL
LIN {X 0,Y 475.879,Z 615.511,A -85,B 0,C 180,E1 -7268.594,E2 -7268.594} C_VEL
LIN {X 0,Y 475.253,Z 634.39,A -85,B 0,C 180,E1 -7271.696,E2 -7271.696} C_VEL
LIN {X 0,Y 475.096,Z 641.553,A -85,B 0,C 180,E1 -7272.867,E2 -7272.867} C_VEL
LIN {X 0,Y 478.404,Z 667.128,A -85,B 0,C 180,E1 -7273.467,E2 -7273.467} C_VEL
LIN {X 0,Y 477.373,Z 753.532,A -85,B 0,C 180,E1 -7274.961,E2 -7274.961} C_VEL
LIN {X 0,Y 476.884,Z 767.476,A -85,B 0,C 180,E1 -7275.382,E2 -7275.382} C_VEL
LIN {X 0,Y 476.371,Z 780.613,A -85,B 0,C 180,E1 -7275.966,E2 -7275.966} C_VEL
LIN {X 0,Y 475.902,Z 792.274,A -85,B 0,C 180,E1 -7276.66,E2 -7276.66} C_VEL
LIN {X 0,Y 475.479,Z 804.235,A -85,B 0,C 180,E1 -7277.564,E2 -7277.564} C_VEL
LIN {X 0,Y 474.962,Z 815.026,A -85,B 0,C 180,E1 -7278.586,E2 -7278.586} C_VEL
LIN {X 0,Y 474.538,Z 825.061,A -85,B 0,C 180,E1 -7279.763,E2 -7279.763} C_VEL
LIN {X 0,Y 474.272,Z 833.936,A -85,B 0,C 180,E1 -7281.049,E2 -7281.049} C_VEL
LIN {X 0,Y 474.089,Z 841.04,A -85,B 0,C 180,E1 -7282.333,E2 -7282.333} C_VEL
LIN {X 0,Y 474.023,Z 846.986,A -85,B 0,C 180,E1 -7283.679,E2 -7283.679} C_VEL
LIN {X 0,Y 473.944,Z 851.21,A -85,B 0,C 180,E1 -7284.896,E2 -7284.896} C_VEL
LIN {X 0,Y 473.979,Z 853.577,A -85,B 0,C 180,E1 -7285.749,E2 -7285.749} C_VEL
LIN {X 0,Y 473.974,Z 855.49,A -85,B 0,C 180,E1 -7286.6,E2 -7286.6} C_VEL
LIN {X 0,Y 473.958,Z 856.92,A -85,B 0,C 180,E1 -7287.451,E2 -7287.451} C_VEL
LIN {X 0,Y 473.925,Z 857.913,A -85,B 0,C 180,E1 -7288.301,E2 -7288.301} C_VEL
LIN {X 0,Y 474.022,Z 858.68,A -85,B 0,C 180,E1 -7290.001,E2 -7290.001} C_VEL
LIN {X 0,Y 473.917,Z 858.392,A -85,B 0,C 180,E1 -7290.85,E2 -7290.85} C_VEL
LIN {X 0,Y 473.952,Z 857.696,A -85,B 0,C 180,E1 -7291.7,E2 -7291.7} C_VEL
LIN {X 0,Y 473.997,Z 856.58,A -85,B 0,C 180,E1 -7292.55,E2 -7292.55} C_VEL
LIN {X 0,Y 474.046,Z 854.074,A -85,B 0,C 180,E1 -7293.826,E2 -7293.826} C_VEL
LIN {X 0,Y 474.077,Z 850.515,A -85,B 0,C 180,E1 -7295.104,E2 -7295.104} C_VEL
LIN {X 0,Y 474.09,Z 845.762,A -85,B 0,C 180,E1 -7296.394,E2 -7296.394} C_VEL
LIN {X 0,Y 474.173,Z 839.822,A -85,B 0,C 180,E1 -7297.666,E2 -7297.666} C_VEL
LIN {X 0,Y 474.296,Z 832.378,A -85,B 0,C 180,E1 -7298.951,E2 -7298.951} C_VEL
LIN {X 0,Y 474.499,Z 824.805,A -85,B 0,C 180,E1 -7300.023,E2 -7300.023} C_VEL
LIN {X 0,Y 474.873,Z 814.643,A -85,B 0,C 180,E1 -7301.201,E2 -7301.201} C_VEL
LIN {X 0,Y 475.201,Z 803.534,A -85,B 0,C 180,E1 -7302.247,E2 -7302.247} C_VEL
LIN {X 0,Y 475.721,Z 791.85,A -85,B 0,C 180,E1 -7303.129,E2 -7303.129} C_VEL
LIN {X 0,Y 476.083,Z 780.216,A -85,B 0,C 180,E1 -7303.826,E2 -7303.826} C_VEL
LIN {X 0,Y 476.593,Z 766.156,A -85,B 0,C 180,E1 -7304.464,E2 -7304.464} C_VEL
LIN {X 0,Y 477.041,Z 752.677,A -85,B 0,C 180,E1 -7304.887,E2 -7304.887} C_VEL
LIN {X 0,Y 477.313,Z 732.514,A -85,B 0,C 180,E1 -7305.26,E2 -7305.26} C_VEL
LIN {X 0,Y 477.875,Z 665.67,A -85,B 0,C 180,E1 -7306.378,E2 -7306.378} C_VEL
LIN {X 0,Y 476.511,Z 654.498,A -85,B 0,C 180,E1 -7306.625,E2 -7306.625} C_VEL
LIN {X 0,Y 475.014,Z 633.553,A -85,B 0,C 180,E1 -7307.074,E2 -7307.074} C_VEL
LIN {X 0,Y 475.242,Z 611.9,A -85,B 0,C 180,E1 -7310.336,E2 -7310.336} C_VEL
LIN {X 0,Y 475.47,Z 590.505,A -85,B 0,C 180,E1 -7313.589,E2 -7313.589} C_VEL
LIN {X 0,Y 475.666,Z 569.857,A -85,B 0,C 180,E1 -7316.785,E2 -7316.785} C_VEL
LIN {X 0,Y 475.839,Z 552.746,A -85,B 0,C 180,E1 -7319.501,E2 -7319.501} C_VEL
LIN {X 0,Y 475.739,Z 547.305,A -85,B 0,C 180,E1 -7320.387,E2 -7320.387} C_VEL
LIN {X 0,Y 474.739,Z 541.352,A -85,B 0,C 180,E1 -7321.425,E2 -7321.425} C_VEL
LIN {X 0,Y 474.637,Z 541.362,A -85,B 0,C 180,E1 -7324.241,E2 -7324.241} C_VEL
LIN {X 0,Y 474.595,Z 541.366,A -85,B 0,C 180,E1 -7327.384,E2 -7327.384} C_VEL
LIN {X 0,Y 474.632,Z 541.359,A -85,B 0,C 180,E1 -7329.648,E2 -7329.648} C_VEL
LIN {X 0,Y 474.611,Z 541.368,A -85,B 0,C 180,E1 -7332.935,E2 -7332.935} C_VEL
LIN {X 0,Y 474.614,Z 541.362,A -85,B 0,C 180,E1 -7335.895,E2 -7335.895} C_VEL
LIN {X 0,Y 474.633,Z 541.364,A -85,B 0,C 180,E1 -7339.041,E2 -7339.041} C_VEL
LIN {X 0,Y 474.615,Z 541.362,A -85,B 0,C 180,E1 -7341.704,E2 -7341.704} C_VEL
LIN {X 0,Y 474.629,Z 541.365,A -85,B 0,C 180,E1 -7344.726,E2 -7344.726} C_VEL
LIN {X 0,Y 474.64,Z 541.359,A -85,B 0,C 180,E1 -7347.788,E2 -7347.788} C_VEL
LIN {X 0,Y 474.629,Z 541.364,A -85,B 0,C 180,E1 -7350.884,E2 -7350.884} C_VEL
LIN {X 0,Y 474.665,Z 541.359,A -85,B 0,C 180,E1 -7353.628,E2 -7353.628} C_VEL
LIN {X 0,Y 474.64,Z 541.365,A -85,B 0,C 180,E1 -7356.641,E2 -7356.641} C_VEL
LIN {X 0,Y 474.659,Z 541.362,A -85,B 0,C 180,E1 -7360.089,E2 -7360.089} C_VEL
LIN {X 0,Y 474.661,Z 541.363,A -85,B 0,C 180,E1 -7362.054,E2 -7362.054} C_VEL
LIN {X 0,Y 479.268,Z 554.081,A -85,B 0,C 180,E1 -7362.441,E2 -7362.441} C_VEL
LIN {X 0,Y 479.255,Z 588.244,A -85,B 0,C 180,E1 -7362.985,E2 -7362.985} C_VEL
LIN {X 0,Y 479.199,Z 603.077,A -85,B 0,C 180,E1 -7363.396,E2 -7363.396} C_VEL
LIN {X 0,Y 479.086,Z 616.491,A -85,B 0,C 180,E1 -7363.925,E2 -7363.925} C_VEL
LIN {X 0,Y 478.766,Z 629.128,A -85,B 0,C 180,E1 -7364.569,E2 -7364.569} C_VEL
LIN {X 0,Y 478.324,Z 642.452,A -85,B 0,C 180,E1 -7365.426,E2 -7365.426} C_VEL
LIN {X 0,Y 477.835,Z 655.792,A -85,B 0,C 180,E1 -7366.497,E2 -7366.497} C_VEL
LIN {X 0,Y 477.308,Z 667.743,A -85,B 0,C 180,E1 -7367.672,E2 -7367.672} C_VEL
LIN {X 0,Y 476.641,Z 678.541,A -85,B 0,C 180,E1 -7368.949,E2 -7368.949} C_VEL
LIN {X 0,Y 476.251,Z 687.54,A -85,B 0,C 180,E1 -7370.229,E2 -7370.229} C_VEL
LIN {X 0,Y 475.749,Z 696.668,A -85,B 0,C 180,E1 -7371.794,E2 -7371.794} C_VEL
LIN {X 0,Y 475.338,Z 703.446,A -85,B 0,C 180,E1 -7373.207,E2 -7373.207} C_VEL
LIN {X 0,Y 474.951,Z 710.077,A -85,B 0,C 180,E1 -7374.906,E2 -7374.906} C_VEL
LIN {X 0,Y 474.738,Z 715.192,A -85,B 0,C 180,E1 -7376.605,E2 -7376.605} C_VEL
LIN {X 0,Y 474.498,Z 718.991,A -85,B 0,C 180,E1 -7378.302,E2 -7378.302} C_VEL
LIN {X 0,Y 474.377,Z 721.547,A -85,B 0,C 180,E1 -7380,E2 -7380} C_VEL
LIN {X 0,Y 474.319,Z 722.931,A -85,B 0,C 180,E1 -7381.698,E2 -7381.698} C_VEL
LIN {X 0,Y 474.422,Z 723.176,A -85,B 0,C 180,E1 -7382.547,E2 -7382.547} C_VEL
LIN {X 0,Y 474.305,Z 722.863,A -85,B 0,C 180,E1 -7384.248,E2 -7384.248} C_VEL
LIN {X 0,Y 474.413,Z 721.375,A -85,B 0,C 180,E1 -7385.952,E2 -7385.952} C_VEL
LIN {X 0,Y 474.487,Z 718.716,A -85,B 0,C 180,E1 -7387.66,E2 -7387.66} C_VEL
LIN {X 0,Y 474.668,Z 714.784,A -85,B 0,C 180,E1 -7389.373,E2 -7389.373} C_VEL
LIN {X 0,Y 474.808,Z 709.511,A -85,B 0,C 180,E1 -7391.094,E2 -7391.094} C_VEL
LIN {X 0,Y 475.164,Z 702.722,A -85,B 0,C 180,E1 -7392.818,E2 -7392.818} C_VEL
LIN {X 0,Y 475.586,Z 695.333,A -85,B 0,C 180,E1 -7394.331,E2 -7394.331} C_VEL
LIN {X 0,Y 476.05,Z 686.39,A -85,B 0,C 180,E1 -7395.85,E2 -7395.85} C_VEL
LIN {X 0,Y 476.647,Z 675.521,A -85,B 0,C 180,E1 -7397.372,E2 -7397.372} C_VEL
LIN {X 0,Y 477.245,Z 664.196,A -85,B 0,C 180,E1 -7398.68,E2 -7398.68} C_VEL
LIN {X 0,Y 477.834,Z 651.613,A -85,B 0,C 180,E1 -7399.884,E2 -7399.884} C_VEL
LIN {X 0,Y 478.39,Z 639.114,A -85,B 0,C 180,E1 -7400.87,E2 -7400.87} C_VEL
LIN {X 0,Y 478.92,Z 625.405,A -85,B 0,C 180,E1 -7401.748,E2 -7401.748} C_VEL
LIN {X 0,Y 479.397,Z 611.447,A -85,B 0,C 180,E1 -7402.454,E2 -7402.454} C_VEL
LIN {X 0,Y 479.621,Z 596.743,A -85,B 0,C 180,E1 -7403.023,E2 -7403.023} C_VEL
LIN {X 0,Y 479.779,Z 581.726,A -85,B 0,C 180,E1 -7403.426,E2 -7403.426} C_VEL
LIN {X 0,Y 479.82,Z 555.438,A -85,B 0,C 180,E1 -7403.875,E2 -7403.875} C_VEL
LIN {X 0,Y 474.702,Z 541.695,A -85,B 0,C 180,E1 -7404.301,E2 -7404.301} C_VEL
LIN {X 0,Y 474.648,Z 541.363,A -85,B 0,C 180,E1 -7404.344,E2 -7404.344} C_VEL
LIN {X 0,Y 474.683,Z 541.354,A -85,B 0,C 180,E1 -7407.334,E2 -7407.334} C_VEL
LIN {X 0,Y 474.607,Z 541.367,A -85,B 0,C 180,E1 -7410.23,E2 -7410.23} C_VEL
LIN {X 0,Y 474.644,Z 541.356,A -85,B 0,C 180,E1 -7413.219,E2 -7413.219} C_VEL
LIN {X 0,Y 474.59,Z 541.369,A -85,B 0,C 180,E1 -7416.323,E2 -7416.323} C_VEL
LIN {X 0,Y 474.629,Z 541.359,A -85,B 0,C 180,E1 -7419.647,E2 -7419.647} C_VEL
LIN {X 0,Y 474.615,Z 541.361,A -85,B 0,C 180,E1 -7422.934,E2 -7422.934} C_VEL
LIN {X 0,Y 474.606,Z 541.364,A -85,B 0,C 180,E1 -7425.894,E2 -7425.894} C_VEL
LIN {X 0,Y 474.628,Z 541.359,A -85,B 0,C 180,E1 -7429.04,E2 -7429.04} C_VEL
LIN {X 0,Y 474.61,Z 541.361,A -85,B 0,C 180,E1 -7431.703,E2 -7431.703} C_VEL
LIN {X 0,Y 474.626,Z 541.364,A -85,B 0,C 180,E1 -7434.725,E2 -7434.725} C_VEL
LIN {X 0,Y 474.636,Z 541.357,A -85,B 0,C 180,E1 -7437.787,E2 -7437.787} C_VEL
LIN {X 0,Y 474.623,Z 541.363,A -85,B 0,C 180,E1 -7440.884,E2 -7440.884} C_VEL
LIN {X 0,Y 474.659,Z 541.357,A -85,B 0,C 180,E1 -7442.237,E2 -7442.237} C_VEL
LIN {X 0,Y 474.02,Z 541.442,A -85,B 0,C 180,E1 -7442.946,E2 -7442.946} C_VEL
LIN {X 0,Y 471.139,Z 541.798,A -85,B 0,C 180,E1 -7444.095,E2 -7444.095} C_VEL
LIN {X 0,Y 468.69,Z 542.102,A -85,B 0,C 180,E1 -7445.022,E2 -7445.022} C_VEL
LIN {X 0,Y 467.648,Z 542.228,A -85,B 0,C 180,E1 -7445.739,E2 -7445.739} C_VEL
LIN {X 0,Y 467.57,Z 542.238,A -85,B 0,C 180,E1 -7445.982,E2 -7445.982} C_VEL
LIN {X 0,Y 467.623,Z 542.231,A -85,B 0,C 180,E1 -7449.777,E2 -7449.777} C_VEL
LIN {X 0,Y 467.608,Z 542.237,A -85,B 0,C 180,E1 -7452.506,E2 -7452.506} C_VEL
LIN {X 0,Y 467.606,Z 542.237,A -85,B 0,C 180,E1 -7455.196,E2 -7455.196} C_VEL
LIN {X 0,Y 467.655,Z 542.227,A -85,B 0,C 180,E1 -7457.854,E2 -7457.854} C_VEL
LIN {X 0,Y 467.68,Z 542.227,A -85,B 0,C 180,E1 -7461.357,E2 -7461.357} C_VEL
LIN {X 0,Y 467.742,Z 542.216,A -85,B 0,C 180,E1 -7463.962,E2 -7463.962} C_VEL
LIN {X 0,Y 467.858,Z 542.205,A -85,B 0,C 180,E1 -7467.417,E2 -7467.417} C_VEL
LIN {X 0,Y 467.881,Z 542.199,A -85,B 0,C 180,E1 -7469.999,E2 -7469.999} C_VEL
LIN {X 0,Y 467.859,Z 542.203,A -85,B 0,C 180,E1 -7472.582,E2 -7472.582} C_VEL
LIN {X 0,Y 467.733,Z 542.217,A -85,B 0,C 180,E1 -7476.037,E2 -7476.037} C_VEL
LIN {X 0,Y 467.679,Z 542.225,A -85,B 0,C 180,E1 -7478.642,E2 -7478.642} C_VEL
LIN {X 0,Y 467.689,Z 542.222,A -85,B 0,C 180,E1 -7482.378,E2 -7482.378} C_VEL
LIN {X 0,Y 467.646,Z 542.23,A -85,B 0,C 180,E1 -7485.885,E2 -7485.885} C_VEL
LIN {X 0,Y 467.621,Z 542.237,A -85,B 0,C 180,E1 -7489.307,E2 -7489.307} C_VEL
LIN {X 0,Y 467.533,Z 542.244,A -85,B 0,C 180,E1 -7492.073,E2 -7492.073} C_VEL
LIN {X 0,Y 467.6,Z 542.234,A -85,B 0,C 180,E1 -7494.887,E2 -7494.887} C_VEL
LIN {X 0,Y 467.624,Z 542.238,A -85,B 0,C 180,E1 -7497.768,E2 -7497.768} C_VEL
LIN {X 0,Y 467.569,Z 542.238,A -85,B 0,C 180,E1 -7501.046,E2 -7501.046} C_VEL
LIN {X 0,Y 467.585,Z 542.238,A -85,B 0,C 180,E1 -7504.242,E2 -7504.242} C_VEL
LIN {X 0,Y 467.546,Z 542.241,A -85,B 0,C 180,E1 -7507.187,E2 -7507.187} C_VEL
LIN {X 0,Y 467.59,Z 542.238,A -85,B 0,C 180,E1 -7510.262,E2 -7510.262} C_VEL
LIN {X 0,Y 467.581,Z 542.237,A -85,B 0,C 180,E1 -7512.567,E2 -7512.567} C_VEL
LIN {X 0,Y 467.565,Z 542.238,A -85,B 0,C 180,E1 -7515.053,E2 -7515.053} C_VEL
LIN {X 0,Y 467.619,Z 542.233,A -85,B 0,C 180,E1 -7517.444,E2 -7517.444} C_VEL
LIN {X 0,Y 467.619,Z 542.232,A -85,B 0,C 180,E1 -7520.859,E2 -7520.859} C_VEL
LIN {X 0,Y 467.558,Z 542.246,A -85,B 0,C 180,E1 -7524.26,E2 -7524.26} C_VEL
LIN {X 0,Y 467.577,Z 542.238,A -85,B 0,C 180,E1 -7527.321,E2 -7527.321} C_VEL
LIN {X 0,Y 467.582,Z 542.246,A -85,B 0,C 180,E1 -7527.962,E2 -7527.962} C_VEL
LIN {X 0,Y 472.238,Z 555.276,A -85,B 0,C 180,E1 -7528.359,E2 -7528.359} C_VEL
LIN {X 0,Y 471.765,Z 600.152,A -85,B 0,C 180,E1 -7529.102,E2 -7529.102} C_VEL
LIN {X 0,Y 471.603,Z 614.317,A -85,B 0,C 180,E1 -7529.503,E2 -7529.503} C_VEL
LIN {X 0,Y 471.374,Z 627.857,A -85,B 0,C 180,E1 -7530.059,E2 -7530.059} C_VEL
LIN {X 0,Y 470.932,Z 640.475,A -85,B 0,C 180,E1 -7530.742,E2 -7530.742} C_VEL
LIN {X 0,Y 470.473,Z 652.582,A -85,B 0,C 180,E1 -7531.575,E2 -7531.575} C_VEL
LIN {X 0,Y 469.946,Z 664.782,A -85,B 0,C 180,E1 -7532.622,E2 -7532.622} C_VEL
LIN {X 0,Y 469.377,Z 675.485,A -85,B 0,C 180,E1 -7533.743,E2 -7533.743} C_VEL
LIN {X 0,Y 468.884,Z 685.015,A -85,B 0,C 180,E1 -7534.949,E2 -7534.949} C_VEL
LIN {X 0,Y 468.42,Z 694.161,A -85,B 0,C 180,E1 -7536.352,E2 -7536.352} C_VEL
LIN {X 0,Y 468.067,Z 701.467,A -85,B 0,C 180,E1 -7537.721,E2 -7537.721} C_VEL
LIN {X 0,Y 467.695,Z 708.382,A -85,B 0,C 180,E1 -7539.321,E2 -7539.321} C_VEL
LIN {X 0,Y 467.521,Z 713.045,A -85,B 0,C 180,E1 -7540.688,E2 -7540.688} C_VEL
LIN {X 0,Y 467.375,Z 716.673,A -85,B 0,C 180,E1 -7542.046,E2 -7542.046} C_VEL
LIN {X 0,Y 467.213,Z 719.395,A -85,B 0,C 180,E1 -7543.393,E2 -7543.393} C_VEL
LIN {X 0,Y 467.127,Z 721.703,A -85,B 0,C 180,E1 -7545.181,E2 -7545.181} C_VEL
LIN {X 0,Y 467.182,Z 722.582,A -85,B 0,C 180,E1 -7546.959,E2 -7546.959} C_VEL
LIN {X 0,Y 467.227,Z 722.051,A -85,B 0,C 180,E1 -7548.724,E2 -7548.724} C_VEL
LIN {X 0,Y 467.275,Z 720.135,A -85,B 0,C 180,E1 -7550.477,E2 -7550.477} C_VEL
LIN {X 0,Y 467.441,Z 716.806,A -85,B 0,C 180,E1 -7552.224,E2 -7552.224} C_VEL
LIN {X 0,Y 467.714,Z 713.308,A -85,B 0,C 180,E1 -7553.53,E2 -7553.53} C_VEL
LIN {X 0,Y 467.902,Z 707.266,A -85,B 0,C 180,E1 -7555.262,E2 -7555.262} C_VEL
LIN {X 0,Y 468.318,Z 700.443,A -85,B 0,C 180,E1 -7556.774,E2 -7556.774} C_VEL
LIN {X 0,Y 468.71,Z 691.979,A -85,B 0,C 180,E1 -7558.282,E2 -7558.282} C_VEL
LIN {X 0,Y 469.303,Z 683.015,A -85,B 0,C 180,E1 -7559.571,E2 -7559.571} C_VEL
LIN {X 0,Y 469.628,Z 674.167,A -85,B 0,C 180,E1 -7560.643,E2 -7560.643} C_VEL
LIN {X 0,Y 470.242,Z 663.409,A -85,B 0,C 180,E1 -7561.713,E2 -7561.713} C_VEL
LIN {X 0,Y 470.742,Z 651.586,A -85,B 0,C 180,E1 -7562.674,E2 -7562.674} C_VEL
LIN {X 0,Y 471.089,Z 640.211,A -85,B 0,C 180,E1 -7563.422,E2 -7563.422} C_VEL
LIN {X 0,Y 471.465,Z 626.646,A -85,B 0,C 180,E1 -7564.114,E2 -7564.114} C_VEL
LIN {X 0,Y 471.646,Z 613.133,A -85,B 0,C 180,E1 -7564.621,E2 -7564.621} C_VEL
LIN {X 0,Y 471.697,Z 598.872,A -85,B 0,C 180,E1 -7564.969,E2 -7564.969} C_VEL
LIN {X 0,Y 471.878,Z 554.011,A -85,B 0,C 180,E1 -7565.68,E2 -7565.68} C_VEL
LIN {X 0,Y 467.738,Z 542.224,A -85,B 0,C 180,E1 -7566.065,E2 -7566.065} C_VEL
LIN {X 0,Y 467.678,Z 542.228,A -85,B 0,C 180,E1 -7568.643,E2 -7568.643} C_VEL
LIN {X 0,Y 467.68,Z 542.23,A -85,B 0,C 180,E1 -7572.145,E2 -7572.145} C_VEL
LIN {X 0,Y 467.646,Z 542.236,A -85,B 0,C 180,E1 -7575.886,E2 -7575.886} C_VEL
LIN {X 0,Y 467.621,Z 542.24,A -85,B 0,C 180,E1 -7579.308,E2 -7579.308} C_VEL
LIN {X 0,Y 467.534,Z 542.246,A -85,B 0,C 180,E1 -7582.074,E2 -7582.074} C_VEL
LIN {X 0,Y 467.601,Z 542.237,A -85,B 0,C 180,E1 -7584.888,E2 -7584.888} C_VEL
LIN {X 0,Y 467.626,Z 542.233,A -85,B 0,C 180,E1 -7587.769,E2 -7587.769} C_VEL
LIN {X 0,Y 467.57,Z 542.239,A -85,B 0,C 180,E1 -7591.047,E2 -7591.047} C_VEL
LIN {X 0,Y 467.587,Z 542.232,A -85,B 0,C 180,E1 -7594.243,E2 -7594.243} C_VEL
LIN {X 0,Y 467.547,Z 542.243,A -85,B 0,C 180,E1 -7597.187,E2 -7597.187} C_VEL
LIN {X 0,Y 467.577,Z 542.237,A -85,B 0,C 180,E1 -7600.265,E2 -7600.265} C_VEL
LIN {X 0,Y 467.585,Z 542.236,A -85,B 0,C 180,E1 -7602.568,E2 -7602.568} C_VEL
LIN {X 0,Y 467.57,Z 542.244,A -85,B 0,C 180,E1 -7605.054,E2 -7605.054} C_VEL
LIN {X 0,Y 467.588,Z 542.24,A -85,B 0,C 180,E1 -7607.441,E2 -7607.441} C_VEL
LIN {X 0,Y 467.582,Z 542.243,A -85,B 0,C 180,E1 -7610.856,E2 -7610.856} C_VEL
LIN {X 0,Y 467.562,Z 542.244,A -85,B 0,C 180,E1 -7614.261,E2 -7614.261} C_VEL
LIN {X 0,Y 467.615,Z 542.254,A -85,B 0,C 180,E1 -7615.288,E2 -7615.288} C_VEL
LIN {X 0,Y 470.887,Z 557.386,A -85,B 0,C 180,E1 -7618.291,E2 -7618.291} C_VEL
LIN {X 0,Y 471.35,Z 561.372,A -85,B 0,C 180,E1 -7619.043,E2 -7619.043} C_VEL
LIN {X 0,Y 470.458,Z 578.687,A -85,B 0,C 180,E1 -7622.104,E2 -7622.104} C_VEL
LIN {X 0,Y 469.56,Z 597.962,A -85,B 0,C 180,E1 -7625.435,E2 -7625.435} C_VEL
LIN {X 0,Y 468.813,Z 618.471,A -85,B 0,C 180,E1 -7628.914,E2 -7628.914} C_VEL
LIN {X 0,Y 468.118,Z 638.791,A -85,B 0,C 180,E1 -7632.301,E2 -7632.301} C_VEL
LIN {X 0,Y 468.055,Z 640.371,A -85,B 0,C 180,E1 -7632.563,E2 -7632.563} C_VEL
LIN {X 0,Y 471.669,Z 668.305,A -85,B 0,C 180,E1 -7633.224,E2 -7633.224} C_VEL
LIN {X 0,Y 470.517,Z 752.739,A -85,B 0,C 180,E1 -7634.737,E2 -7634.737} C_VEL
LIN {X 0,Y 470.002,Z 766.563,A -85,B 0,C 180,E1 -7635.163,E2 -7635.163} C_VEL
LIN {X 0,Y 469.479,Z 778.629,A -85,B 0,C 180,E1 -7635.7,E2 -7635.7} C_VEL
LIN {X 0,Y 468.963,Z 791.276,A -85,B 0,C 180,E1 -7636.458,E2 -7636.458} C_VEL
LIN {X 0,Y 468.43,Z 802.952,A -85,B 0,C 180,E1 -7637.351,E2 -7637.351} C_VEL
LIN {X 0,Y 468.014,Z 813.018,A -85,B 0,C 180,E1 -7638.304,E2 -7638.304} C_VEL
LIN {X 0,Y 467.579,Z 822.401,A -85,B 0,C 180,E1 -7639.39,E2 -7639.39} C_VEL
LIN {X 0,Y 467.274,Z 831.573,A -85,B 0,C 180,E1 -7640.696,E2 -7640.696} C_VEL
LIN {X 0,Y 467.064,Z 838.99,A -85,B 0,C 180,E1 -7642,E2 -7642} C_VEL
LIN {X 0,Y 466.938,Z 845.34,A -85,B 0,C 180,E1 -7643.408,E2 -7643.408} C_VEL
LIN {X 0,Y 466.934,Z 848.885,A -85,B 0,C 180,E1 -7644.386,E2 -7644.386} C_VEL
LIN {X 0,Y 466.925,Z 852.611,A -85,B 0,C 180,E1 -7645.684,E2 -7645.684} C_VEL
LIN {X 0,Y 466.93,Z 854.525,A -85,B 0,C 180,E1 -7646.549,E2 -7646.549} C_VEL
LIN {X 0,Y 466.912,Z 855.954,A -85,B 0,C 180,E1 -7647.412,E2 -7647.412} C_VEL
LIN {X 0,Y 466.887,Z 856.94,A -85,B 0,C 180,E1 -7648.275,E2 -7648.275} C_VEL
LIN {X 0,Y 467.008,Z 857.697,A -85,B 0,C 180,E1 -7650.001,E2 -7650.001} C_VEL
LIN {X 0,Y 466.886,Z 857.395,A -85,B 0,C 180,E1 -7650.863,E2 -7650.863} C_VEL
LIN {X 0,Y 466.92,Z 856.678,A -85,B 0,C 180,E1 -7651.726,E2 -7651.726} C_VEL
LIN {X 0,Y 466.958,Z 855.546,A -85,B 0,C 180,E1 -7652.588,E2 -7652.588} C_VEL
LIN {X 0,Y 467.009,Z 853.008,A -85,B 0,C 180,E1 -7653.884,E2 -7653.884} C_VEL
LIN {X 0,Y 467.025,Z 849.408,A -85,B 0,C 180,E1 -7655.181,E2 -7655.181} C_VEL
LIN {X 0,Y 467.056,Z 843.687,A -85,B 0,C 180,E1 -7656.716,E2 -7656.716} C_VEL
LIN {X 0,Y 467.141,Z 837.501,A -85,B 0,C 180,E1 -7658,E2 -7658} C_VEL
LIN {X 0,Y 467.28,Z 829.686,A -85,B 0,C 180,E1 -7659.305,E2 -7659.305} C_VEL
LIN {X 0,Y 467.571,Z 820.019,A -85,B 0,C 180,E1 -7660.611,E2 -7660.611} C_VEL
LIN {X 0,Y 467.93,Z 810.101,A -85,B 0,C 180,E1 -7661.699,E2 -7661.699} C_VEL
LIN {X 0,Y 468.303,Z 798.698,A -85,B 0,C 180,E1 -7662.713,E2 -7662.713} C_VEL
LIN {X 0,Y 468.748,Z 788.705,A -85,B 0,C 180,E1 -7663.439,E2 -7663.439} C_VEL
LIN {X 0,Y 469.221,Z 776.663,A -85,B 0,C 180,E1 -7664.143,E2 -7664.143} C_VEL
LIN {X 0,Y 469.743,Z 763.281,A -85,B 0,C 180,E1 -7664.735,E2 -7664.735} C_VEL
LIN {X 0,Y 470.242,Z 749.052,A -85,B 0,C 180,E1 -7665.162,E2 -7665.162} C_VEL
LIN {X 0,Y 470.587,Z 715.794,A -85,B 0,C 180,E1 -7665.752,E2 -7665.752} C_VEL
LIN {X 0,Y 471.003,Z 666.357,A -85,B 0,C 180,E1 -7666.613,E2 -7666.613} C_VEL
LIN {X 0,Y 469.632,Z 653.047,A -85,B 0,C 180,E1 -7666.911,E2 -7666.911} C_VEL
LIN {X 0,Y 467.922,Z 631.054,A -85,B 0,C 180,E1 -7667.411,E2 -7667.411} C_VEL
LIN {X 0,Y 468.187,Z 609.883,A -85,B 0,C 180,E1 -7670.657,E2 -7670.657} C_VEL
LIN {X 0,Y 468.437,Z 587.483,A -85,B 0,C 180,E1 -7674.132,E2 -7674.132} C_VEL
LIN {X 0,Y 468.624,Z 567.982,A -85,B 0,C 180,E1 -7677.221,E2 -7677.221} C_VEL
LIN {X 0,Y 468.857,Z 550.034,A -85,B 0,C 180,E1 -7680.143,E2 -7680.143} C_VEL
LIN {X 0,Y 467.672,Z 542.232,A -85,B 0,C 180,E1 -7681.525,E2 -7681.525} C_VEL
LIN {X 0,Y 467.57,Z 542.246,A -85,B 0,C 180,E1 -7684.833,E2 -7684.833} C_VEL
LIN {X 0,Y 467.57,Z 542.239,A -85,B 0,C 180,E1 -7688.045,E2 -7688.045} C_VEL
LIN {X 0,Y 467.582,Z 542.24,A -85,B 0,C 180,E1 -7691.277,E2 -7691.277} C_VEL
LIN {X 0,Y 467.555,Z 542.241,A -85,B 0,C 180,E1 -7693.821,E2 -7693.821} C_VEL
LIN {X 0,Y 467.561,Z 542.243,A -85,B 0,C 180,E1 -7696.256,E2 -7696.256} C_VEL
LIN {X 0,Y 467.583,Z 542.242,A -85,B 0,C 180,E1 -7698.723,E2 -7698.723} C_VEL
LIN {X 0,Y 467.57,Z 542.24,A -85,B 0,C 180,E1 -7701.955,E2 -7701.955} C_VEL
LIN {X 0,Y 467.568,Z 542.242,A -85,B 0,C 180,E1 -7705.167,E2 -7705.167} C_VEL
LIN {X 0,Y 467.587,Z 542.241,A -85,B 0,C 180,E1 -7708.26,E2 -7708.26} C_VEL
LIN {X 0,Y 467.581,Z 542.24,A -85,B 0,C 180,E1 -7711.25,E2 -7711.25} C_VEL
LIN {X 0,Y 467.615,Z 542.241,A -85,B 0,C 180,E1 -7714.16,E2 -7714.16} C_VEL
LIN {X 0,Y 467.581,Z 542.243,A -85,B 0,C 180,E1 -7716.996,E2 -7716.996} C_VEL
LIN {X 0,Y 467.627,Z 542.236,A -85,B 0,C 180,E1 -7719.777,E2 -7719.777} C_VEL
LIN {X 0,Y 467.637,Z 542.237,A -85,B 0,C 180,E1 -7721.758,E2 -7721.758} C_VEL
LIN {X 0,Y 469.73,Z 548.043,A -85,B 0,C 180,E1 -7721.946,E2 -7721.946} C_VEL
LIN {X 0,Y 472.615,Z 556.233,A -85,B 0,C 180,E1 -7722.2,E2 -7722.2} C_VEL
LIN {X 0,Y 472.546,Z 588.724,A -85,B 0,C 180,E1 -7722.719,E2 -7722.719} C_VEL
LIN {X 0,Y 472.514,Z 604.033,A -85,B 0,C 180,E1 -7723.141,E2 -7723.141} C_VEL
LIN {X 0,Y 472.383,Z 617.865,A -85,B 0,C 180,E1 -7723.691,E2 -7723.691} C_VEL
LIN {X 0,Y 472.055,Z 630.525,A -85,B 0,C 180,E1 -7724.344,E2 -7724.344} C_VEL
LIN {X 0,Y 471.589,Z 643.864,A -85,B 0,C 180,E1 -7725.214,E2 -7725.214} C_VEL
LIN {X 0,Y 471.101,Z 655.965,A -85,B 0,C 180,E1 -7726.19,E2 -7726.19} C_VEL
LIN {X 0,Y 470.546,Z 668.105,A -85,B 0,C 180,E1 -7727.382,E2 -7727.382} C_VEL
LIN {X 0,Y 469.807,Z 679.828,A -85,B 0,C 180,E1 -7728.786,E2 -7728.786} C_VEL
LIN {X 0,Y 469.372,Z 688.817,A -85,B 0,C 180,E1 -7730.084,E2 -7730.084} C_VEL
LIN {X 0,Y 468.86,Z 697.647,A -85,B 0,C 180,E1 -7731.617,E2 -7731.617} C_VEL
LIN {X 0,Y 468.398,Z 704.703,A -85,B 0,C 180,E1 -7733.106,E2 -7733.106} C_VEL
LIN {X 0,Y 467.988,Z 711.311,A -85,B 0,C 180,E1 -7734.83,E2 -7734.83} C_VEL
LIN {X 0,Y 467.767,Z 716.395,A -85,B 0,C 180,E1 -7736.554,E2 -7736.554} C_VEL
LIN {X 0,Y 467.496,Z 720.153,A -85,B 0,C 180,E1 -7738.277,E2 -7738.277} C_VEL
LIN {X 0,Y 467.364,Z 722.663,A -85,B 0,C 180,E1 -7740,E2 -7740} C_VEL
LIN {X 0,Y 467.328,Z 723.994,A -85,B 0,C 180,E1 -7741.723,E2 -7741.723} C_VEL
LIN {X 0,Y 467.406,Z 724.217,A -85,B 0,C 180,E1 -7742.585,E2 -7742.585} C_VEL
LIN {X 0,Y 467.283,Z 723.849,A -85,B 0,C 180,E1 -7744.312,E2 -7744.312} C_VEL
LIN {X 0,Y 467.406,Z 722.303,A -85,B 0,C 180,E1 -7746.041,E2 -7746.041} C_VEL
LIN {X 0,Y 467.473,Z 719.583,A -85,B 0,C 180,E1 -7747.776,E2 -7747.776} C_VEL
LIN {X 0,Y 467.655,Z 715.592,A -85,B 0,C 180,E1 -7749.515,E2 -7749.515} C_VEL
LIN {X 0,Y 467.845,Z 710.236,A -85,B 0,C 180,E1 -7751.261,E2 -7751.261} C_VEL
LIN {X 0,Y 468.233,Z 703.332,A -85,B 0,C 180,E1 -7753.011,E2 -7753.011} C_VEL
LIN {X 0,Y 468.665,Z 695.858,A -85,B 0,C 180,E1 -7754.547,E2 -7754.547} C_VEL
LIN {X 0,Y 469.157,Z 686.94,A -85,B 0,C 180,E1 -7756.063,E2 -7756.063} C_VEL
LIN {X 0,Y 469.687,Z 677.422,A -85,B 0,C 180,E1 -7757.413,E2 -7757.413} C_VEL
LIN {X 0,Y 470.314,Z 666.255,A -85,B 0,C 180,E1 -7758.74,E2 -7758.74} C_VEL
LIN {X 0,Y 470.963,Z 654.238,A -85,B 0,C 180,E1 -7759.927,E2 -7759.927} C_VEL
LIN {X 0,Y 471.524,Z 641.616,A -85,B 0,C 180,E1 -7760.96,E2 -7760.96} C_VEL
LIN {X 0,Y 472.04,Z 628.255,A -85,B 0,C 180,E1 -7761.852,E2 -7761.852} C_VEL
LIN {X 0,Y 472.548,Z 613.705,A -85,B 0,C 180,E1 -7762.62,E2 -7762.62} C_VEL
LIN {X 0,Y 472.86,Z 598.591,A -85,B 0,C 180,E1 -7763.223,E2 -7763.223} C_VEL
LIN {X 0,Y 473.01,Z 583.181,A -85,B 0,C 180,E1 -7763.651,E2 -7763.651} C_VEL
LIN {X 0,Y 473.003,Z 556.939,A -85,B 0,C 180,E1 -7764.109,E2 -7764.109} C_VEL
LIN {X 0,Y 467.631,Z 542.235,A -85,B 0,C 180,E1 -7764.579,E2 -7764.579} C_VEL
LIN {X 0,Y 467.622,Z 542.238,A -85,B 0,C 180,E1 -7767.768,E2 -7767.768} C_VEL
LIN {X 0,Y 467.569,Z 542.237,A -85,B 0,C 180,E1 -7771.044,E2 -7771.044} C_VEL
LIN {X 0,Y 467.589,Z 542.242,A -85,B 0,C 180,E1 -7774.242,E2 -7774.242} C_VEL
LIN {X 0,Y 467.549,Z 542.24,A -85,B 0,C 180,E1 -7777.186,E2 -7777.186} C_VEL
LIN {X 0,Y 467.578,Z 542.245,A -85,B 0,C 180,E1 -7780.264,E2 -7780.264} C_VEL
LIN {X 0,Y 467.587,Z 542.24,A -85,B 0,C 180,E1 -7782.566,E2 -7782.566} C_VEL
LIN {X 0,Y 467.566,Z 542.238,A -85,B 0,C 180,E1 -7785.052,E2 -7785.052} C_VEL
LIN {X 0,Y 467.589,Z 542.235,A -85,B 0,C 180,E1 -7787.439,E2 -7787.439} C_VEL
LIN {X 0,Y 467.582,Z 542.239,A -85,B 0,C 180,E1 -7790.855,E2 -7790.855} C_VEL
LIN {X 0,Y 467.56,Z 542.244,A -85,B 0,C 180,E1 -7794.26,E2 -7794.26} C_VEL
LIN {X 0,Y 467.581,Z 542.236,A -85,B 0,C 180,E1 -7797.32,E2 -7797.32} C_VEL
LIN {X 0,Y 467.57,Z 542.245,A -85,B 0,C 180,E1 -7800.667,E2 -7800.667} C_VEL
LIN {X 0,Y 467.615,Z 542.233,A -85,B 0,C 180,E1 -7803.199,E2 -7803.199} C_VEL
LIN {X 0,Y 467.57,Z 542.238,A -85,B 0,C 180,E1 -7805.982,E2 -7805.982} C_VEL
LIN {X 0,Y 466.922,Z 542.327,A -85,B 0,C 180,E1 -7806.701,E2 -7806.701} C_VEL
LIN {X 0,Y 464.075,Z 542.676,A -85,B 0,C 180,E1 -7807.869,E2 -7807.869} C_VEL
LIN {X 0,Y 461.659,Z 542.982,A -85,B 0,C 180,E1 -7808.811,E2 -7808.811} C_VEL
LIN {X 0,Y 460.625,Z 543.103,A -85,B 0,C 180,E1 -7809.538,E2 -7809.538} C_VEL
LIN {X 0,Y 460.544,Z 543.112,A -85,B 0,C 180,E1 -7809.785,E2 -7809.785} C_VEL
LIN {X 0,Y 460.558,Z 543.112,A -85,B 0,C 180,E1 -7812.23,E2 -7812.23} C_VEL
LIN {X 0,Y 460.565,Z 543.117,A -85,B 0,C 180,E1 -7814.964,E2 -7814.964} C_VEL
LIN {X 0,Y 460.61,Z 543.108,A -85,B 0,C 180,E1 -7818.559,E2 -7818.559} C_VEL
LIN {X 0,Y 460.693,Z 543.094,A -85,B 0,C 180,E1 -7822.108,E2 -7822.108} C_VEL
LIN {X 0,Y 460.696,Z 543.098,A -85,B 0,C 180,E1 -7824.748,E2 -7824.748} C_VEL
LIN {X 0,Y 460.823,Z 543.082,A -85,B 0,C 180,E1 -7827.377,E2 -7827.377} C_VEL
LIN {X 0,Y 460.852,Z 543.074,A -85,B 0,C 180,E1 -7829.999,E2 -7829.999} C_VEL
LIN {X 0,Y 460.824,Z 543.079,A -85,B 0,C 180,E1 -7832.622,E2 -7832.622} C_VEL
LIN {X 0,Y 460.699,Z 543.093,A -85,B 0,C 180,E1 -7836.13,E2 -7836.13} C_VEL
LIN {X 0,Y 460.626,Z 543.104,A -85,B 0,C 180,E1 -7838.776,E2 -7838.776} C_VEL
LIN {X 0,Y 460.631,Z 543.102,A -85,B 0,C 180,E1 -7842.456,E2 -7842.456} C_VEL
LIN {X 0,Y 460.596,Z 543.108,A -85,B 0,C 180,E1 -7845.997,E2 -7845.997} C_VEL
LIN {X 0,Y 460.568,Z 543.111,A -85,B 0,C 180,E1 -7848.902,E2 -7848.902} C_VEL
LIN {X 0,Y 460.512,Z 543.125,A -85,B 0,C 180,E1 -7851.485,E2 -7851.485} C_VEL
LIN {X 0,Y 460.539,Z 543.114,A -85,B 0,C 180,E1 -7854.332,E2 -7854.332} C_VEL
LIN {X 0,Y 460.58,Z 543.111,A -85,B 0,C 180,E1 -7857.243,E2 -7857.243} C_VEL
LIN {X 0,Y 460.523,Z 543.117,A -85,B 0,C 180,E1 -7860.238,E2 -7860.238} C_VEL
LIN {X 0,Y 460.525,Z 543.118,A -85,B 0,C 180,E1 -7863.324,E2 -7863.324} C_VEL
LIN {X 0,Y 460.474,Z 543.122,A -85,B 0,C 180,E1 -7866.529,E2 -7866.529} C_VEL
LIN {X 0,Y 460.569,Z 543.118,A -85,B 0,C 180,E1 -7869.858,E2 -7869.858} C_VEL
LIN {X 0,Y 460.507,Z 543.117,A -85,B 0,C 180,E1 -7872.9,E2 -7872.9} C_VEL
LIN {X 0,Y 460.518,Z 543.122,A -85,B 0,C 180,E1 -7875.829,E2 -7875.829} C_VEL
LIN {X 0,Y 460.539,Z 543.113,A -85,B 0,C 180,E1 -7878.99,E2 -7878.99} C_VEL
LIN {X 0,Y 460.544,Z 543.113,A -85,B 0,C 180,E1 -7881.269,E2 -7881.269} C_VEL
LIN {X 0,Y 460.509,Z 543.12,A -85,B 0,C 180,E1 -7884.555,E2 -7884.555} C_VEL
LIN {X 0,Y 460.558,Z 543.115,A -85,B 0,C 180,E1 -7887.691,E2 -7887.691} C_VEL
LIN {X 0,Y 465.317,Z 556.298,A -85,B 0,C 180,E1 -7888.114,E2 -7888.114} C_VEL
LIN {X 0,Y 464.953,Z 601.484,A -85,B 0,C 180,E1 -7888.882,E2 -7888.882} C_VEL
LIN {X 0,Y 464.783,Z 615.829,A -85,B 0,C 180,E1 -7889.299,E2 -7889.299} C_VEL
LIN {X 0,Y 464.5,Z 630.116,A -85,B 0,C 180,E1 -7889.905,E2 -7889.905} C_VEL
LIN {X 0,Y 464.065,Z 643.051,A -85,B 0,C 180,E1 -7890.64,E2 -7890.64} C_VEL
LIN {X 0,Y 463.584,Z 654.66,A -85,B 0,C 180,E1 -7891.469,E2 -7891.469} C_VEL
LIN {X 0,Y 463.018,Z 666.833,A -85,B 0,C 180,E1 -7892.545,E2 -7892.545} C_VEL
LIN {X 0,Y 462.445,Z 677.679,A -85,B 0,C 180,E1 -7893.72,E2 -7893.72} C_VEL
LIN {X 0,Y 461.923,Z 687.604,A -85,B 0,C 180,E1 -7895.027,E2 -7895.027} C_VEL
LIN {X 0,Y 461.466,Z 695.831,A -85,B 0,C 180,E1 -7896.338,E2 -7896.338} C_VEL
LIN {X 0,Y 461.085,Z 703.523,A -85,B 0,C 180,E1 -7897.837,E2 -7897.837} C_VEL
LIN {X 0,Y 460.681,Z 710.187,A -85,B 0,C 180,E1 -7899.459,E2 -7899.459} C_VEL
LIN {X 0,Y 460.457,Z 715.511,A -85,B 0,C 180,E1 -7901.138,E2 -7901.138} C_VEL
LIN {X 0,Y 460.326,Z 718.213,A -85,B 0,C 180,E1 -7902.221,E2 -7902.221} C_VEL
LIN {X 0,Y 460.166,Z 721.443,A -85,B 0,C 180,E1 -7904.044,E2 -7904.044} C_VEL
LIN {X 0,Y 460.112,Z 723.2,A -85,B 0,C 180,E1 -7905.854,E2 -7905.854} C_VEL
LIN {X 0,Y 460.178,Z 723.544,A -85,B 0,C 180,E1 -7907.655,E2 -7907.655} C_VEL
LIN {X 0,Y 460.208,Z 722.516,A -85,B 0,C 180,E1 -7909.441,E2 -7909.441} C_VEL
LIN {X 0,Y 460.325,Z 720.055,A -85,B 0,C 180,E1 -7911.218,E2 -7911.218} C_VEL
LIN {X 0,Y 460.624,Z 716.131,A -85,B 0,C 180,E1 -7912.989,E2 -7912.989} C_VEL
LIN {X 0,Y 460.843,Z 710.71,A -85,B 0,C 180,E1 -7914.75,E2 -7914.75} C_VEL
LIN {X 0,Y 461.136,Z 705.468,A -85,B 0,C 180,E1 -7916.068,E2 -7916.068} C_VEL
LIN {X 0,Y 461.54,Z 697.971,A -85,B 0,C 180,E1 -7917.6,E2 -7917.6} C_VEL
LIN {X 0,Y 462.051,Z 690.058,A -85,B 0,C 180,E1 -7918.911,E2 -7918.911} C_VEL
LIN {X 0,Y 462.58,Z 680.489,A -85,B 0,C 180,E1 -7920.218,E2 -7920.218} C_VEL
LIN {X 0,Y 463.097,Z 669.778,A -85,B 0,C 180,E1 -7921.414,E2 -7921.414} C_VEL
LIN {X 0,Y 463.715,Z 657.769,A -85,B 0,C 180,E1 -7922.498,E2 -7922.498} C_VEL
LIN {X 0,Y 464.209,Z 645.844,A -85,B 0,C 180,E1 -7923.364,E2 -7923.364} C_VEL
LIN {X 0,Y 464.596,Z 632.586,A -85,B 0,C 180,E1 -7924.121,E2 -7924.121} C_VEL
LIN {X 0,Y 464.845,Z 618.461,A -85,B 0,C 180,E1 -7924.716,E2 -7924.716} C_VEL
LIN {X 0,Y 464.912,Z 604.316,A -85,B 0,C 180,E1 -7925.123,E2 -7925.123} C_VEL
LIN {X 0,Y 465.191,Z 555.663,A -85,B 0,C 180,E1 -7925.93,E2 -7925.93} C_VEL
LIN {X 0,Y 460.702,Z 543.101,A -85,B 0,C 180,E1 -7926.35,E2 -7926.35} C_VEL
LIN {X 0,Y 460.625,Z 543.107,A -85,B 0,C 180,E1 -7928.777,E2 -7928.777} C_VEL
LIN {X 0,Y 460.631,Z 543.107,A -85,B 0,C 180,E1 -7932.457,E2 -7932.457} C_VEL
LIN {X 0,Y 460.597,Z 543.113,A -85,B 0,C 180,E1 -7935.998,E2 -7935.998} C_VEL
LIN {X 0,Y 460.568,Z 543.115,A -85,B 0,C 180,E1 -7938.903,E2 -7938.903} C_VEL
LIN {X 0,Y 460.513,Z 543.123,A -85,B 0,C 180,E1 -7941.486,E2 -7941.486} C_VEL
LIN {X 0,Y 460.54,Z 543.115,A -85,B 0,C 180,E1 -7944.333,E2 -7944.333} C_VEL
LIN {X 0,Y 460.582,Z 543.113,A -85,B 0,C 180,E1 -7947.244,E2 -7947.244} C_VEL
LIN {X 0,Y 460.525,Z 543.112,A -85,B 0,C 180,E1 -7950.239,E2 -7950.239} C_VEL
LIN {X 0,Y 460.527,Z 543.119,A -85,B 0,C 180,E1 -7953.325,E2 -7953.325} C_VEL
LIN {X 0,Y 460.475,Z 543.12,A -85,B 0,C 180,E1 -7956.53,E2 -7956.53} C_VEL
LIN {X 0,Y 460.557,Z 543.113,A -85,B 0,C 180,E1 -7959.86,E2 -7959.86} C_VEL
LIN {X 0,Y 460.516,Z 543.12,A -85,B 0,C 180,E1 -7962.902,E2 -7962.902} C_VEL
LIN {X 0,Y 460.51,Z 543.119,A -85,B 0,C 180,E1 -7965.831,E2 -7965.831} C_VEL
LIN {X 0,Y 460.53,Z 543.116,A -85,B 0,C 180,E1 -7968.989,E2 -7968.989} C_VEL
LIN {X 0,Y 460.526,Z 543.124,A -85,B 0,C 180,E1 -7971.268,E2 -7971.268} C_VEL
LIN {X 0,Y 460.566,Z 543.119,A -85,B 0,C 180,E1 -7974.921,E2 -7974.921} C_VEL
LIN {X 0,Y 460.576,Z 543.175,A -85,B 0,C 180,E1 -7975.042,E2 -7975.042} C_VEL
LIN {X 0,Y 463.811,Z 558.1,A -85,B 0,C 180,E1 -7978.055,E2 -7978.055} C_VEL
LIN {X 0,Y 464.438,Z 561.856,A -85,B 0,C 180,E1 -7978.784,E2 -7978.784} C_VEL
LIN {X 0,Y 463.579,Z 577.83,A -85,B 0,C 180,E1 -7981.658,E2 -7981.658} C_VEL
LIN {X 0,Y 462.654,Z 595.818,A -85,B 0,C 180,E1 -7984.829,E2 -7984.829} C_VEL
LIN {X 0,Y 461.932,Z 613.849,A -85,B 0,C 180,E1 -7987.951,E2 -7987.951} C_VEL
LIN {X 0,Y 461.187,Z 633.74,A -85,B 0,C 180,E1 -7991.337,E2 -7991.337} C_VEL
LIN {X 0,Y 461.039,Z 639.131,A -85,B 0,C 180,E1 -7992.25,E2 -7992.25} C_VEL
LIN {X 0,Y 464.898,Z 668.929,A -85,B 0,C 180,E1 -7992.973,E2 -7992.973} C_VEL
LIN {X 0,Y 463.683,Z 751.821,A -85,B 0,C 180,E1 -7994.506,E2 -7994.506} C_VEL
LIN {X 0,Y 463.125,Z 765.53,A -85,B 0,C 180,E1 -7994.938,E2 -7994.938} C_VEL
LIN {X 0,Y 462.573,Z 777.562,A -85,B 0,C 180,E1 -7995.482,E2 -7995.482} C_VEL
LIN {X 0,Y 461.964,Z 790.204,A -85,B 0,C 180,E1 -7996.249,E2 -7996.249} C_VEL
LIN {X 0,Y 461.438,Z 801.892,A -85,B 0,C 180,E1 -7997.156,E2 -7997.156} C_VEL
LIN {X 0,Y 460.939,Z 811.966,A -85,B 0,C 180,E1 -7998.122,E2 -7998.122} C_VEL
LIN {X 0,Y 460.542,Z 821.378,A -85,B 0,C 180,E1 -7999.226,E2 -7999.226} C_VEL
LIN {X 0,Y 460.206,Z 830.565,A -85,B 0,C 180,E1 -8000.552,E2 -8000.552} C_VEL
LIN {X 0,Y 460.012,Z 838,A -85,B 0,C 180,E1 -8001.876,E2 -8001.876} C_VEL
LIN {X 0,Y 459.862,Z 843.022,A -85,B 0,C 180,E1 -8002.978,E2 -8002.978} C_VEL
LIN {X 0,Y 459.88,Z 847.915,A -85,B 0,C 180,E1 -8004.3,E2 -8004.3} C_VEL
LIN {X 0,Y 459.874,Z 851.644,A -85,B 0,C 180,E1 -8005.618,E2 -8005.618} C_VEL
LIN {X 0,Y 459.887,Z 853.561,A -85,B 0,C 180,E1 -8006.496,E2 -8006.496} C_VEL
LIN {X 0,Y 459.866,Z 854.984,A -85,B 0,C 180,E1 -8007.373,E2 -8007.373} C_VEL
LIN {X 0,Y 459.848,Z 855.967,A -85,B 0,C 180,E1 -8008.249,E2 -8008.249} C_VEL
LIN {X 0,Y 459.992,Z 856.713,A -85,B 0,C 180,E1 -8010.001,E2 -8010.001} C_VEL
LIN {X 0,Y 459.855,Z 856.391,A -85,B 0,C 180,E1 -8010.876,E2 -8010.876} C_VEL
LIN {X 0,Y 459.886,Z 855.662,A -85,B 0,C 180,E1 -8011.752,E2 -8011.752} C_VEL
LIN {X 0,Y 459.918,Z 854.517,A -85,B 0,C 180,E1 -8012.628,E2 -8012.628} C_VEL
LIN {X 0,Y 459.972,Z 851.951,A -85,B 0,C 180,E1 -8013.943,E2 -8013.943} C_VEL
LIN {X 0,Y 459.974,Z 848.314,A -85,B 0,C 180,E1 -8015.26,E2 -8015.26} C_VEL
LIN {X 0,Y 459.991,Z 842.913,A -85,B 0,C 180,E1 -8016.728,E2 -8016.728} C_VEL
LIN {X 0,Y 460.077,Z 836.302,A -85,B 0,C 180,E1 -8018.124,E2 -8018.124} C_VEL
LIN {X 0,Y 460.241,Z 828.437,A -85,B 0,C 180,E1 -8019.449,E2 -8019.449} C_VEL
LIN {X 0,Y 460.531,Z 818.721,A -85,B 0,C 180,E1 -8020.775,E2 -8020.775} C_VEL
LIN {X 0,Y 460.945,Z 808.77,A -85,B 0,C 180,E1 -8021.879,E2 -8021.879} C_VEL
LIN {X 0,Y 461.266,Z 798.605,A -85,B 0,C 180,E1 -8022.805,E2 -8022.805} C_VEL
LIN {X 0,Y 461.69,Z 787.284,A -85,B 0,C 180,E1 -8023.648,E2 -8023.648} C_VEL
LIN {X 0,Y 462.331,Z 774.237,A -85,B 0,C 180,E1 -8024.414,E2 -8024.414} C_VEL
LIN {X 0,Y 462.883,Z 760.438,A -85,B 0,C 180,E1 -8025.015,E2 -8025.015} C_VEL
LIN {X 0,Y 463.418,Z 745.743,A -85,B 0,C 180,E1 -8025.447,E2 -8025.447} C_VEL
LIN {X 0,Y 464.253,Z 667.456,A -85,B 0,C 180,E1 -8026.849,E2 -8026.849} C_VEL
LIN {X 0,Y 462.863,Z 653.657,A -85,B 0,C 180,E1 -8027.166,E2 -8027.166} C_VEL
LIN {X 0,Y 460.864,Z 628.58,A -85,B 0,C 180,E1 -8027.758,E2 -8027.758} C_VEL
LIN {X 0,Y 461.153,Z 607.926,A -85,B 0,C 180,E1 -8030.987,E2 -8030.987} C_VEL
LIN {X 0,Y 461.363,Z 585.573,A -85,B 0,C 180,E1 -8034.526,E2 -8034.526} C_VEL
LIN {X 0,Y 461.574,Z 567.646,A -85,B 0,C 180,E1 -8037.426,E2 -8037.426} C_VEL
LIN {X 0,Y 461.836,Z 551.272,A -85,B 0,C 180,E1 -8040.145,E2 -8040.145} C_VEL
LIN {X 0,Y 460.634,Z 543.108,A -85,B 0,C 180,E1 -8041.615,E2 -8041.615} C_VEL
LIN {X 0,Y 460.537,Z 543.12,A -85,B 0,C 180,E1 -8044.506,E2 -8044.506} C_VEL
LIN {X 0,Y 460.506,Z 543.12,A -85,B 0,C 180,E1 -8047.623,E2 -8047.623} C_VEL
LIN {X 0,Y 460.546,Z 543.115,A -85,B 0,C 180,E1 -8050.269,E2 -8050.269} C_VEL
LIN {X 0,Y 460.502,Z 543.121,A -85,B 0,C 180,E1 -8053.376,E2 -8053.376} C_VEL
LIN {X 0,Y 460.505,Z 543.123,A -85,B 0,C 180,E1 -8056.625,E2 -8056.625} C_VEL
LIN {X 0,Y 460.546,Z 543.115,A -85,B 0,C 180,E1 -8059.731,E2 -8059.731} C_VEL
LIN {X 0,Y 460.504,Z 543.123,A -85,B 0,C 180,E1 -8062.524,E2 -8062.524} C_VEL
LIN {X 0,Y 460.55,Z 543.115,A -85,B 0,C 180,E1 -8065.624,E2 -8065.624} C_VEL
LIN {X 0,Y 460.542,Z 543.121,A -85,B 0,C 180,E1 -8068.744,E2 -8068.744} C_VEL
LIN {X 0,Y 460.586,Z 543.116,A -85,B 0,C 180,E1 -8072.254,E2 -8072.254} C_VEL
LIN {X 0,Y 460.564,Z 543.12,A -85,B 0,C 180,E1 -8074.705,E2 -8074.705} C_VEL
LIN {X 0,Y 460.516,Z 543.122,A -85,B 0,C 180,E1 -8077.571,E2 -8077.571} C_VEL
LIN {X 0,Y 460.573,Z 543.117,A -85,B 0,C 180,E1 -8080.384,E2 -8080.384} C_VEL
LIN {X 0,Y 460.599,Z 543.112,A -85,B 0,C 180,E1 -8081.449,E2 -8081.449} C_VEL
LIN {X 0,Y 462.749,Z 548.87,A -85,B 0,C 180,E1 -8081.644,E2 -8081.644} C_VEL
LIN {X 0,Y 465.874,Z 557.201,A -85,B 0,C 180,E1 -8081.917,E2 -8081.917} C_VEL
LIN {X 0,Y 465.898,Z 590.404,A -85,B 0,C 180,E1 -8082.465,E2 -8082.465} C_VEL
LIN {X 0,Y 465.859,Z 605.201,A -85,B 0,C 180,E1 -8082.879,E2 -8082.879} C_VEL
LIN {X 0,Y 465.687,Z 619.343,A -85,B 0,C 180,E1 -8083.449,E2 -8083.449} C_VEL
LIN {X 0,Y 465.358,Z 631.932,A -85,B 0,C 180,E1 -8084.113,E2 -8084.113} C_VEL
LIN {X 0,Y 464.869,Z 645.274,A -85,B 0,C 180,E1 -8084.995,E2 -8084.995} C_VEL
LIN {X 0,Y 464.336,Z 658.581,A -85,B 0,C 180,E1 -8086.097,E2 -8086.097} C_VEL
LIN {X 0,Y 463.777,Z 669.511,A -85,B 0,C 180,E1 -8087.195,E2 -8087.195} C_VEL
LIN {X 0,Y 462.983,Z 681.216,A -85,B 0,C 180,E1 -8088.618,E2 -8088.618} C_VEL
LIN {X 0,Y 462.517,Z 690.165,A -85,B 0,C 180,E1 -8089.936,E2 -8089.936} C_VEL
LIN {X 0,Y 461.95,Z 699.346,A -85,B 0,C 180,E1 -8091.575,E2 -8091.575} C_VEL
LIN {X 0,Y 461.461,Z 705.959,A -85,B 0,C 180,E1 -8093.001,E2 -8093.001} C_VEL
LIN {X 0,Y 461.025,Z 712.542,A -85,B 0,C 180,E1 -8094.752,E2 -8094.752} C_VEL
LIN {X 0,Y 460.793,Z 717.598,A -85,B 0,C 180,E1 -8096.502,E2 -8096.502} C_VEL
LIN {X 0,Y 460.495,Z 721.323,A -85,B 0,C 180,E1 -8098.25,E2 -8098.25} C_VEL
LIN {X 0,Y 460.353,Z 723.791,A -85,B 0,C 180,E1 -8100,E2 -8100} C_VEL
LIN {X 0,Y 460.333,Z 725.072,A -85,B 0,C 180,E1 -8101.749,E2 -8101.749} C_VEL
LIN {X 0,Y 460.247,Z 725.213,A -85,B 0,C 180,E1 -8103.501,E2 -8103.501} C_VEL
LIN {X 0,Y 460.378,Z 724.175,A -85,B 0,C 180,E1 -8105.255,E2 -8105.255} C_VEL
LIN {X 0,Y 460.417,Z 721.733,A -85,B 0,C 180,E1 -8107.165,E2 -8107.165} C_VEL
LIN {X 0,Y 460.58,Z 718.557,A -85,B 0,C 180,E1 -8108.777,E2 -8108.777} C_VEL
LIN {X 0,Y 460.737,Z 713.816,A -85,B 0,C 180,E1 -8110.547,E2 -8110.547} C_VEL
LIN {X 0,Y 461.084,Z 707.606,A -85,B 0,C 180,E1 -8112.321,E2 -8112.321} C_VEL
LIN {X 0,Y 461.539,Z 699.725,A -85,B 0,C 180,E1 -8114.101,E2 -8114.101} C_VEL
LIN {X 0,Y 462.032,Z 691.238,A -85,B 0,C 180,E1 -8115.664,E2 -8115.664} C_VEL
LIN {X 0,Y 462.56,Z 682.552,A -85,B 0,C 180,E1 -8117.006,E2 -8117.006} C_VEL
LIN {X 0,Y 463.157,Z 672.196,A -85,B 0,C 180,E1 -8118.352,E2 -8118.352} C_VEL
LIN {X 0,Y 463.837,Z 660.499,A -85,B 0,C 180,E1 -8119.618,E2 -8119.618} C_VEL
LIN {X 0,Y 464.374,Z 648.355,A -85,B 0,C 180,E1 -8120.717,E2 -8120.717} C_VEL
LIN {X 0,Y 465.023,Z 634.57,A -85,B 0,C 180,E1 -8121.732,E2 -8121.732} C_VEL
LIN {X 0,Y 465.578,Z 620.204,A -85,B 0,C 180,E1 -8122.574,E2 -8122.574} C_VEL
LIN {X 0,Y 465.997,Z 605.94,A -85,B 0,C 180,E1 -8123.221,E2 -8123.221} C_VEL
LIN {X 0,Y 466.148,Z 590.825,A -85,B 0,C 180,E1 -8123.726,E2 -8123.726} C_VEL
LIN {X 0,Y 466.289,Z 574.225,A -85,B 0,C 180,E1 -8124.078,E2 -8124.078} C_VEL
LIN {X 0,Y 466.22,Z 558.428,A -85,B 0,C 180,E1 -8124.352,E2 -8124.352} C_VEL
LIN {X 0,Y 460.605,Z 543.397,A -85,B 0,C 180,E1 -8124.848,E2 -8124.848} C_VEL
LIN {X 0,Y 460.55,Z 543.116,A -85,B 0,C 180,E1 -8124.892,E2 -8124.892} C_VEL
LIN {X 0,Y 460.554,Z 543.118,A -85,B 0,C 180,E1 -8128.232,E2 -8128.232} C_VEL
LIN {X 0,Y 460.522,Z 543.116,A -85,B 0,C 180,E1 -8131.282,E2 -8131.282} C_VEL
LIN {X 0,Y 460.533,Z 543.117,A -85,B 0,C 180,E1 -8134.505,E2 -8134.505} C_VEL
LIN {X 0,Y 460.502,Z 543.119,A -85,B 0,C 180,E1 -8137.623,E2 -8137.623} C_VEL
LIN {X 0,Y 460.542,Z 543.121,A -85,B 0,C 180,E1 -8140.269,E2 -8140.269} C_VEL
LIN {X 0,Y 460.498,Z 543.118,A -85,B 0,C 180,E1 -8143.375,E2 -8143.375} C_VEL
LIN {X 0,Y 460.498,Z 543.123,A -85,B 0,C 180,E1 -8146.624,E2 -8146.624} C_VEL
LIN {X 0,Y 460.542,Z 543.114,A -85,B 0,C 180,E1 -8149.73,E2 -8149.73} C_VEL
LIN {X 0,Y 460.526,Z 543.123,A -85,B 0,C 180,E1 -8152.519,E2 -8152.519} C_VEL
LIN {X 0,Y 460.547,Z 543.112,A -85,B 0,C 180,E1 -8155.623,E2 -8155.623} C_VEL
LIN {X 0,Y 460.536,Z 543.12,A -85,B 0,C 180,E1 -8158.744,E2 -8158.744} C_VEL
LIN {X 0,Y 460.588,Z 543.11,A -85,B 0,C 180,E1 -8162.252,E2 -8162.252} C_VEL
LIN {X 0,Y 460.558,Z 543.119,A -85,B 0,C 180,E1 -8164.705,E2 -8164.705} C_VEL
LIN {X 0,Y 460.511,Z 543.117,A -85,B 0,C 180,E1 -8167.571,E2 -8167.571} C_VEL
LIN {X 0,Y 460.544,Z 543.112,A -85,B 0,C 180,E1 -8169.785,E2 -8169.785} C_VEL
LIN {X 0,Y 459.876,Z 543.203,A -85,B 0,C 180,E1 -8170.514,E2 -8170.514} C_VEL
LIN {X 0,Y 457.002,Z 543.557,A -85,B 0,C 180,E1 -8171.699,E2 -8171.699} C_VEL
LIN {X 0,Y 454.592,Z 543.86,A -85,B 0,C 180,E1 -8172.655,E2 -8172.655} C_VEL
LIN {X 0,Y 453.592,Z 543.981,A -85,B 0,C 180,E1 -8173.394,E2 -8173.394} C_VEL
LIN {X 0,Y 453.528,Z 543.987,A -85,B 0,C 180,E1 -8173.644,E2 -8173.644} C_VEL
LIN {X 0,Y 453.51,Z 543.993,A -85,B 0,C 180,E1 -8176.558,E2 -8176.558} C_VEL
LIN {X 0,Y 453.531,Z 543.99,A -85,B 0,C 180,E1 -8179.283,E2 -8179.283} C_VEL
LIN {X 0,Y 453.692,Z 543.968,A -85,B 0,C 180,E1 -8182.479,E2 -8182.479} C_VEL
LIN {X 0,Y 453.669,Z 543.972,A -85,B 0,C 180,E1 -8184.666,E2 -8184.666} C_VEL
LIN {X 0,Y 453.764,Z 543.962,A -85,B 0,C 180,E1 -8187.336,E2 -8187.336} C_VEL
LIN {X 0,Y 453.822,Z 543.95,A -85,B 0,C 180,E1 -8189.999,E2 -8189.999} C_VEL
LIN {X 0,Y 453.764,Z 543.959,A -85,B 0,C 180,E1 -8192.663,E2 -8192.663} C_VEL
LIN {X 0,Y 453.667,Z 543.969,A -85,B 0,C 180,E1 -8196.225,E2 -8196.225} C_VEL
LIN {X 0,Y 453.59,Z 543.982,A -85,B 0,C 180,E1 -8198.913,E2 -8198.913} C_VEL
LIN {X 0,Y 453.598,Z 543.978,A -85,B 0,C 180,E1 -8202.55,E2 -8202.55} C_VEL
LIN {X 0,Y 453.541,Z 543.985,A -85,B 0,C 180,E1 -8206.195,E2 -8206.195} C_VEL
LIN {X 0,Y 453.517,Z 543.99,A -85,B 0,C 180,E1 -8209.041,E2 -8209.041} C_VEL
LIN {X 0,Y 453.473,Z 543.998,A -85,B 0,C 180,E1 -8211.836,E2 -8211.836} C_VEL
LIN {X 0,Y 453.51,Z 543.989,A -85,B 0,C 180,E1 -8214.734,E2 -8214.734} C_VEL
LIN {X 0,Y 453.534,Z 543.99,A -85,B 0,C 180,E1 -8217.961,E2 -8217.961} C_VEL
LIN {X 0,Y 453.479,Z 543.993,A -85,B 0,C 180,E1 -8220.759,E2 -8220.759} C_VEL
LIN {X 0,Y 453.473,Z 544,A -85,B 0,C 180,E1 -8223.912,E2 -8223.912} C_VEL
LIN {X 0,Y 453.466,Z 543.995,A -85,B 0,C 180,E1 -8227.188,E2 -8227.188} C_VEL
LIN {X 0,Y 453.523,Z 543.99,A -85,B 0,C 180,E1 -8229.445,E2 -8229.445} C_VEL
LIN {X 0,Y 453.473,Z 544.002,A -85,B 0,C 180,E1 -8231.935,E2 -8231.935} C_VEL
LIN {X 0,Y 453.488,Z 543.994,A -85,B 0,C 180,E1 -8235.47,E2 -8235.47} C_VEL
LIN {X 0,Y 453.491,Z 543.997,A -85,B 0,C 180,E1 -8238.211,E2 -8238.211} C_VEL
LIN {X 0,Y 453.53,Z 543.987,A -85,B 0,C 180,E1 -8240.787,E2 -8240.787} C_VEL
LIN {X 0,Y 453.452,Z 544.001,A -85,B 0,C 180,E1 -8243.918,E2 -8243.918} C_VEL
LIN {X 0,Y 453.482,Z 543.994,A -85,B 0,C 180,E1 -8247.152,E2 -8247.152} C_VEL
LIN {X 0,Y 453.506,Z 543.991,A -85,B 0,C 180,E1 -8247.429,E2 -8247.429} C_VEL
LIN {X 0,Y 458.647,Z 558.135,A -85,B 0,C 180,E1 -8247.89,E2 -8247.89} C_VEL
LIN {X 0,Y 458.17,Z 603.09,A -85,B 0,C 180,E1 -8248.671,E2 -8248.671} C_VEL
LIN {X 0,Y 457.987,Z 616.842,A -85,B 0,C 180,E1 -8249.081,E2 -8249.081} C_VEL
LIN {X 0,Y 457.679,Z 630.848,A -85,B 0,C 180,E1 -8249.681,E2 -8249.681} C_VEL
LIN {X 0,Y 457.24,Z 643.613,A -85,B 0,C 180,E1 -8250.411,E2 -8250.411} C_VEL
LIN {X 0,Y 456.724,Z 655.797,A -85,B 0,C 180,E1 -8251.294,E2 -8251.294} C_VEL
LIN {X 0,Y 456.14,Z 667.549,A -85,B 0,C 180,E1 -8252.345,E2 -8252.345} C_VEL
LIN {X 0,Y 455.508,Z 678.994,A -85,B 0,C 180,E1 -8253.601,E2 -8253.601} C_VEL
LIN {X 0,Y 454.997,Z 688.446,A -85,B 0,C 180,E1 -8254.864,E2 -8254.864} C_VEL
LIN {X 0,Y 454.482,Z 697.265,A -85,B 0,C 180,E1 -8256.294,E2 -8256.294} C_VEL
LIN {X 0,Y 454.117,Z 704.452,A -85,B 0,C 180,E1 -8257.718,E2 -8257.718} C_VEL
LIN {X 0,Y 453.734,Z 710.313,A -85,B 0,C 180,E1 -8259.13,E2 -8259.13} C_VEL
LIN {X 0,Y 453.53,Z 715.153,A -85,B 0,C 180,E1 -8260.586,E2 -8260.586} C_VEL
LIN {X 0,Y 453.335,Z 718.659,A -85,B 0,C 180,E1 -8261.938,E2 -8261.938} C_VEL
LIN {X 0,Y 453.173,Z 722.147,A -85,B 0,C 180,E1 -8263.791,E2 -8263.791} C_VEL
LIN {X 0,Y 453.106,Z 724.076,A -85,B 0,C 180,E1 -8265.631,E2 -8265.631} C_VEL
LIN {X 0,Y 453.149,Z 724.586,A -85,B 0,C 180,E1 -8267.46,E2 -8267.46} C_VEL
LIN {X 0,Y 453.18,Z 723.722,A -85,B 0,C 180,E1 -8269.275,E2 -8269.275} C_VEL
LIN {X 0,Y 453.327,Z 721.472,A -85,B 0,C 180,E1 -8271.082,E2 -8271.082} C_VEL
LIN {X 0,Y 453.609,Z 717.721,A -85,B 0,C 180,E1 -8272.88,E2 -8272.88} C_VEL
LIN {X 0,Y 453.855,Z 712.451,A -85,B 0,C 180,E1 -8274.669,E2 -8274.669} C_VEL
LIN {X 0,Y 454.162,Z 707.372,A -85,B 0,C 180,E1 -8276.007,E2 -8276.007} C_VEL
LIN {X 0,Y 454.602,Z 700.043,A -85,B 0,C 180,E1 -8277.564,E2 -8277.564} C_VEL
LIN {X 0,Y 455.077,Z 692.34,A -85,B 0,C 180,E1 -8278.894,E2 -8278.894} C_VEL
LIN {X 0,Y 455.687,Z 683.009,A -85,B 0,C 180,E1 -8280.221,E2 -8280.221} C_VEL
LIN {X 0,Y 456.201,Z 672.682,A -85,B 0,C 180,E1 -8281.435,E2 -8281.435} C_VEL
LIN {X 0,Y 456.828,Z 661.089,A -85,B 0,C 180,E1 -8282.535,E2 -8282.535} C_VEL
LIN {X 0,Y 457.398,Z 649.654,A -85,B 0,C 180,E1 -8283.414,E2 -8283.414} C_VEL
LIN {X 0,Y 457.751,Z 637.18,A -85,B 0,C 180,E1 -8284.183,E2 -8284.183} C_VEL
LIN {X 0,Y 458.058,Z 623.699,A -85,B 0,C 180,E1 -8284.814,E2 -8284.814} C_VEL
LIN {X 0,Y 458.224,Z 610.529,A -85,B 0,C 180,E1 -8285.253,E2 -8285.253} C_VEL
LIN {X 0,Y 458.213,Z 596.036,A -85,B 0,C 180,E1 -8285.556,E2 -8285.556} C_VEL
LIN {X 0,Y 458.468,Z 557.19,A -85,B 0,C 180,E1 -8286.195,E2 -8286.195} C_VEL
LIN {X 0,Y 453.649,Z 544.058,A -85,B 0,C 180,E1 -8286.645,E2 -8286.645} C_VEL
LIN {X 0,Y 453.589,Z 543.985,A -85,B 0,C 180,E1 -8288.914,E2 -8288.914} C_VEL
LIN {X 0,Y 453.598,Z 543.983,A -85,B 0,C 180,E1 -8292.551,E2 -8292.551} C_VEL
LIN {X 0,Y 453.541,Z 543.99,A -85,B 0,C 180,E1 -8296.196,E2 -8296.196} C_VEL
LIN {X 0,Y 453.518,Z 543.994,A -85,B 0,C 180,E1 -8299.042,E2 -8299.042} C_VEL
LIN {X 0,Y 453.474,Z 544,A -85,B 0,C 180,E1 -8301.837,E2 -8301.837} C_VEL
LIN {X 0,Y 453.512,Z 543.991,A -85,B 0,C 180,E1 -8304.735,E2 -8304.735} C_VEL
LIN {X 0,Y 453.536,Z 543.986,A -85,B 0,C 180,E1 -8307.962,E2 -8307.962} C_VEL
LIN {X 0,Y 453.481,Z 543.991,A -85,B 0,C 180,E1 -8310.76,E2 -8310.76} C_VEL
LIN {X 0,Y 453.475,Z 543.991,A -85,B 0,C 180,E1 -8313.913,E2 -8313.913} C_VEL
LIN {X 0,Y 453.468,Z 543.996,A -85,B 0,C 180,E1 -8317.189,E2 -8317.189} C_VEL
LIN {X 0,Y 453.515,Z 543.992,A -85,B 0,C 180,E1 -8319.448,E2 -8319.448} C_VEL
LIN {X 0,Y 453.467,Z 543.999,A -85,B 0,C 180,E1 -8322.995,E2 -8322.995} C_VEL
LIN {X 0,Y 453.465,Z 543.997,A -85,B 0,C 180,E1 -8325.78,E2 -8325.78} C_VEL
LIN {X 0,Y 453.478,Z 543.993,A -85,B 0,C 180,E1 -8328.21,E2 -8328.21} C_VEL
LIN {X 0,Y 453.51,Z 543.995,A -85,B 0,C 180,E1 -8330.792,E2 -8330.792} C_VEL
LIN {X 0,Y 453.457,Z 544.002,A -85,B 0,C 180,E1 -8333.918,E2 -8333.918} C_VEL
LIN {X 0,Y 453.525,Z 544.042,A -85,B 0,C 180,E1 -8334.778,E2 -8334.778} C_VEL
LIN {X 0,Y 456.708,Z 558.826,A -85,B 0,C 180,E1 -8337.819,E2 -8337.819} C_VEL
LIN {X 0,Y 457.509,Z 563.629,A -85,B 0,C 180,E1 -8338.764,E2 -8338.764} C_VEL
LIN {X 0,Y 456.501,Z 581.328,A -85,B 0,C 180,E1 -8341.995,E2 -8341.995} C_VEL
LIN {X 0,Y 455.486,Z 601.253,A -85,B 0,C 180,E1 -8345.555,E2 -8345.555} C_VEL
LIN {X 0,Y 454.676,Z 620.55,A -85,B 0,C 180,E1 -8348.939,E2 -8348.939} C_VEL
LIN {X 0,Y 454.051,Z 637.723,A -85,B 0,C 180,E1 -8351.909,E2 -8351.909} C_VEL
LIN {X 0,Y 458.114,Z 670.381,A -85,B 0,C 180,E1 -8352.738,E2 -8352.738} C_VEL
LIN {X 0,Y 456.831,Z 750.777,A -85,B 0,C 180,E1 -8354.268,E2 -8354.268} C_VEL
LIN {X 0,Y 456.26,Z 764.429,A -85,B 0,C 180,E1 -8354.706,E2 -8354.706} C_VEL
LIN {X 0,Y 455.693,Z 776.455,A -85,B 0,C 180,E1 -8355.258,E2 -8355.258} C_VEL
LIN {X 0,Y 455.018,Z 789.107,A -85,B 0,C 180,E1 -8356.035,E2 -8356.035} C_VEL
LIN {X 0,Y 454.453,Z 801.073,A -85,B 0,C 180,E1 -8356.978,E2 -8356.978} C_VEL
LIN {X 0,Y 453.975,Z 810.911,A -85,B 0,C 180,E1 -8357.937,E2 -8357.937} C_VEL
LIN {X 0,Y 453.493,Z 820.331,A -85,B 0,C 180,E1 -8359.057,E2 -8359.057} C_VEL
LIN {X 0,Y 453.144,Z 829.534,A -85,B 0,C 180,E1 -8360.403,E2 -8360.403} C_VEL
LIN {X 0,Y 452.939,Z 836.984,A -85,B 0,C 180,E1 -8361.749,E2 -8361.749} C_VEL
LIN {X 0,Y 452.791,Z 843.108,A -85,B 0,C 180,E1 -8363.132,E2 -8363.132} C_VEL
LIN {X 0,Y 452.823,Z 846.926,A -85,B 0,C 180,E1 -8364.211,E2 -8364.211} C_VEL
LIN {X 0,Y 452.826,Z 850.664,A -85,B 0,C 180,E1 -8365.55,E2 -8365.55} C_VEL
LIN {X 0,Y 452.845,Z 852.583,A -85,B 0,C 180,E1 -8366.441,E2 -8366.441} C_VEL
LIN {X 0,Y 452.82,Z 854.009,A -85,B 0,C 180,E1 -8367.332,E2 -8367.332} C_VEL
LIN {X 0,Y 452.809,Z 854.991,A -85,B 0,C 180,E1 -8368.222,E2 -8368.222} C_VEL
LIN {X 0,Y 452.975,Z 855.726,A -85,B 0,C 180,E1 -8370.001,E2 -8370.001} C_VEL
LIN {X 0,Y 452.823,Z 855.394,A -85,B 0,C 180,E1 -8370.89,E2 -8370.89} C_VEL
LIN {X 0,Y 452.852,Z 854.65,A -85,B 0,C 180,E1 -8371.779,E2 -8371.779} C_VEL
LIN {X 0,Y 452.879,Z 853.484,A -85,B 0,C 180,E1 -8372.669,E2 -8372.669} C_VEL
LIN {X 0,Y 452.932,Z 850.889,A -85,B 0,C 180,E1 -8374.004,E2 -8374.004} C_VEL
LIN {X 0,Y 452.905,Z 847.218,A -85,B 0,C 180,E1 -8375.343,E2 -8375.343} C_VEL
LIN {X 0,Y 452.941,Z 842.091,A -85,B 0,C 180,E1 -8376.758,E2 -8376.758} C_VEL
LIN {X 0,Y 453.029,Z 835.132,A -85,B 0,C 180,E1 -8378.251,E2 -8378.251} C_VEL
LIN {X 0,Y 453.176,Z 827.214,A -85,B 0,C 180,E1 -8379.597,E2 -8379.597} C_VEL
LIN {X 0,Y 453.482,Z 817.455,A -85,B 0,C 180,E1 -8380.944,E2 -8380.944} C_VEL
LIN {X 0,Y 453.947,Z 807.484,A -85,B 0,C 180,E1 -8382.065,E2 -8382.065} C_VEL
LIN {X 0,Y 454.192,Z 798.798,A -85,B 0,C 180,E1 -8382.879,E2 -8382.879} C_VEL
LIN {X 0,Y 454.662,Z 789.192,A -85,B 0,C 180,E1 -8383.635,E2 -8383.635} C_VEL
LIN {X 0,Y 455.228,Z 777.068,A -85,B 0,C 180,E1 -8384.416,E2 -8384.416} C_VEL
LIN {X 0,Y 455.824,Z 763.455,A -85,B 0,C 180,E1 -8385.081,E2 -8385.081} C_VEL
LIN {X 0,Y 456.408,Z 750.176,A -85,B 0,C 180,E1 -8385.548,E2 -8385.548} C_VEL
LIN {X 0,Y 456.735,Z 735.3,A -85,B 0,C 180,E1 -8385.88,E2 -8385.88} C_VEL
LIN {X 0,Y 457.449,Z 667.93,A -85,B 0,C 180,E1 -8387.113,E2 -8387.113} C_VEL
LIN {X 0,Y 456.076,Z 653.562,A -85,B 0,C 180,E1 -8387.451,E2 -8387.451} C_VEL
LIN {X 0,Y 454.179,Z 629.933,A -85,B 0,C 180,E1 -8388.014,E2 -8388.014} C_VEL
LIN {X 0,Y 453.807,Z 626.047,A -85,B 0,C 180,E1 -8388.131,E2 -8388.131} C_VEL
LIN {X 0,Y 454.062,Z 605.956,A -85,B 0,C 180,E1 -8391.33,E2 -8391.33} C_VEL
LIN {X 0,Y 454.271,Z 585.165,A -85,B 0,C 180,E1 -8394.691,E2 -8394.691} C_VEL
LIN {X 0,Y 454.538,Z 567.339,A -85,B 0,C 180,E1 -8397.637,E2 -8397.637} C_VEL
LIN {X 0,Y 454.805,Z 551.541,A -85,B 0,C 180,E1 -8400.322,E2 -8400.322} C_VEL
LIN {X 0,Y 453.588,Z 543.986,A -85,B 0,C 180,E1 -8401.711,E2 -8401.711} C_VEL
LIN {X 0,Y 453.485,Z 544,A -85,B 0,C 180,E1 -8404.989,E2 -8404.989} C_VEL
LIN {X 0,Y 453.469,Z 543.997,A -85,B 0,C 180,E1 -8408.312,E2 -8408.312} C_VEL
LIN {X 0,Y 453.498,Z 543.995,A -85,B 0,C 180,E1 -8410.609,E2 -8410.609} C_VEL
LIN {X 0,Y 453.459,Z 544,A -85,B 0,C 180,E1 -8413.244,E2 -8413.244} C_VEL
LIN {X 0,Y 453.471,Z 543.996,A -85,B 0,C 180,E1 -8415.779,E2 -8415.779} C_VEL
LIN {X 0,Y 453.484,Z 543.997,A -85,B 0,C 180,E1 -8418.209,E2 -8418.209} C_VEL
LIN {X 0,Y 453.514,Z 543.994,A -85,B 0,C 180,E1 -8420.791,E2 -8420.791} C_VEL
LIN {X 0,Y 453.458,Z 543.999,A -85,B 0,C 180,E1 -8423.917,E2 -8423.917} C_VEL
LIN {X 0,Y 453.487,Z 543.996,A -85,B 0,C 180,E1 -8427.151,E2 -8427.151} C_VEL
LIN {X 0,Y 453.48,Z 543.999,A -85,B 0,C 180,E1 -8430.268,E2 -8430.268} C_VEL
LIN {X 0,Y 453.511,Z 543.995,A -85,B 0,C 180,E1 -8433.294,E2 -8433.294} C_VEL
LIN {X 0,Y 453.508,Z 543.998,A -85,B 0,C 180,E1 -8436.239,E2 -8436.239} C_VEL
LIN {X 0,Y 453.487,Z 543.998,A -85,B 0,C 180,E1 -8439.117,E2 -8439.117} C_VEL
LIN {X 0,Y 453.556,Z 543.99,A -85,B 0,C 180,E1 -8441.092,E2 -8441.092} C_VEL
LIN {X 0,Y 454.454,Z 546.695,A -85,B 0,C 180,E1 -8441.206,E2 -8441.206} C_VEL
LIN {X 0,Y 459.219,Z 558.762,A -85,B 0,C 180,E1 -8441.64,E2 -8441.64} C_VEL
LIN {X 0,Y 459.219,Z 592.214,A -85,B 0,C 180,E1 -8442.201,E2 -8442.201} C_VEL
LIN {X 0,Y 459.223,Z 606.882,A -85,B 0,C 180,E1 -8442.622,E2 -8442.622} C_VEL
LIN {X 0,Y 459.012,Z 621.02,A -85,B 0,C 180,E1 -8443.202,E2 -8443.202} C_VEL
LIN {X 0,Y 458.673,Z 633.593,A -85,B 0,C 180,E1 -8443.875,E2 -8443.875} C_VEL
LIN {X 0,Y 458.166,Z 646.838,A -85,B 0,C 180,E1 -8444.77,E2 -8444.77} C_VEL
LIN {X 0,Y 457.602,Z 660.046,A -85,B 0,C 180,E1 -8445.888,E2 -8445.888} C_VEL
LIN {X 0,Y 457.023,Z 669.89,A -85,B 0,C 180,E1 -8446.89,E2 -8446.89} C_VEL
LIN {X 0,Y 456.327,Z 680.956,A -85,B 0,C 180,E1 -8448.225,E2 -8448.225} C_VEL
LIN {X 0,Y 455.674,Z 691.537,A -85,B 0,C 180,E1 -8449.783,E2 -8449.783} C_VEL
LIN {X 0,Y 455.075,Z 700.509,A -85,B 0,C 180,E1 -8451.409,E2 -8451.409} C_VEL
LIN {X 0,Y 454.539,Z 707.289,A -85,B 0,C 180,E1 -8452.894,E2 -8452.894} C_VEL
LIN {X 0,Y 454.233,Z 712.274,A -85,B 0,C 180,E1 -8454.228,E2 -8454.228} C_VEL
LIN {X 0,Y 453.91,Z 717.644,A -85,B 0,C 180,E1 -8456.004,E2 -8456.004} C_VEL
LIN {X 0,Y 453.61,Z 720.818,A -85,B 0,C 180,E1 -8457.336,E2 -8457.336} C_VEL
LIN {X 0,Y 453.39,Z 723.86,A -85,B 0,C 180,E1 -8459.111,E2 -8459.111} C_VEL
LIN {X 0,Y 453.346,Z 725.676,A -85,B 0,C 180,E1 -8460.888,E2 -8460.888} C_VEL
LIN {X 0,Y 453.37,Z 726.322,A -85,B 0,C 180,E1 -8462.665,E2 -8462.665} C_VEL
LIN {X 0,Y 453.245,Z 725.834,A -85,B 0,C 180,E1 -8464.446,E2 -8464.446} C_VEL
LIN {X 0,Y 453.39,Z 724.152,A -85,B 0,C 180,E1 -8466.229,E2 -8466.229} C_VEL
LIN {X 0,Y 453.479,Z 721.28,A -85,B 0,C 180,E1 -8468.017,E2 -8468.017} C_VEL
LIN {X 0,Y 453.665,Z 717.122,A -85,B 0,C 180,E1 -8469.811,E2 -8469.811} C_VEL
LIN {X 0,Y 453.905,Z 711.575,A -85,B 0,C 180,E1 -8471.612,E2 -8471.612} C_VEL
LIN {X 0,Y 454.345,Z 704.45,A -85,B 0,C 180,E1 -8473.416,E2 -8473.416} C_VEL
LIN {X 0,Y 454.836,Z 696.742,A -85,B 0,C 180,E1 -8474.999,E2 -8474.999} C_VEL
LIN {X 0,Y 455.361,Z 688.036,A -85,B 0,C 180,E1 -8476.488,E2 -8476.488} C_VEL
LIN {X 0,Y 455.999,Z 677.744,A -85,B 0,C 180,E1 -8477.953,E2 -8477.953} C_VEL
LIN {X 0,Y 456.702,Z 666.171,A -85,B 0,C 180,E1 -8479.32,E2 -8479.32} C_VEL
LIN {X 0,Y 457.364,Z 653.812,A -85,B 0,C 180,E1 -8480.532,E2 -8480.532} C_VEL
LIN {X 0,Y 457.949,Z 642.026,A -85,B 0,C 180,E1 -8481.493,E2 -8481.493} C_VEL
LIN {X 0,Y 458.526,Z 628.226,A -85,B 0,C 180,E1 -8482.412,E2 -8482.412} C_VEL
LIN {X 0,Y 459.048,Z 613.615,A -85,B 0,C 180,E1 -8483.174,E2 -8483.174} C_VEL
LIN {X 0,Y 459.338,Z 598.688,A -85,B 0,C 180,E1 -8483.761,E2 -8483.761} C_VEL
LIN {X 0,Y 459.487,Z 584.231,A -85,B 0,C 180,E1 -8484.158,E2 -8484.158} C_VEL
LIN {X 0,Y 459.551,Z 560.236,A -85,B 0,C 180,E1 -8484.594,E2 -8484.594} C_VEL
LIN {X 0,Y 453.51,Z 543.994,A -85,B 0,C 180,E1 -8485.135,E2 -8485.135} C_VEL
LIN {X 0,Y 453.534,Z 543.994,A -85,B 0,C 180,E1 -8487.959,E2 -8487.959} C_VEL
LIN {X 0,Y 453.467,Z 543.996,A -85,B 0,C 180,E1 -8491.524,E2 -8491.524} C_VEL
LIN {X 0,Y 453.488,Z 543.992,A -85,B 0,C 180,E1 -8494.777,E2 -8494.777} C_VEL
LIN {X 0,Y 453.465,Z 544.001,A -85,B 0,C 180,E1 -8498.311,E2 -8498.311} C_VEL
LIN {X 0,Y 453.494,Z 543.994,A -85,B 0,C 180,E1 -8500.608,E2 -8500.608} C_VEL
LIN {X 0,Y 453.455,Z 543.996,A -85,B 0,C 180,E1 -8503.243,E2 -8503.243} C_VEL
LIN {X 0,Y 453.464,Z 543.996,A -85,B 0,C 180,E1 -8505.778,E2 -8505.778} C_VEL
LIN {X 0,Y 453.479,Z 543.999,A -85,B 0,C 180,E1 -8508.209,E2 -8508.209} C_VEL
LIN {X 0,Y 453.515,Z 543.992,A -85,B 0,C 180,E1 -8510.789,E2 -8510.789} C_VEL
LIN {X 0,Y 453.454,Z 543.997,A -85,B 0,C 180,E1 -8513.917,E2 -8513.917} C_VEL
LIN {X 0,Y 453.482,Z 543.993,A -85,B 0,C 180,E1 -8517.151,E2 -8517.151} C_VEL
LIN {X 0,Y 453.474,Z 543.997,A -85,B 0,C 180,E1 -8520.268,E2 -8520.268} C_VEL
LIN {X 0,Y 453.508,Z 543.99,A -85,B 0,C 180,E1 -8523.294,E2 -8523.294} C_VEL
LIN {X 0,Y 453.503,Z 543.992,A -85,B 0,C 180,E1 -8526.238,E2 -8526.238} C_VEL
LIN {X 0,Y 453.485,Z 543.992,A -85,B 0,C 180,E1 -8529.79,E2 -8529.79} C_VEL
LIN {X 0,Y 453.506,Z 543.997,A -85,B 0,C 180,E1 -8532.875,E2 -8532.875} C_VEL
LIN {X 0,Y 453.528,Z 543.987,A -85,B 0,C 180,E1 -8533.644,E2 -8533.644} C_VEL
LIN {X 0,Y 452.913,Z 544.067,A -85,B 0,C 180,E1 -8534.385,E2 -8534.385} C_VEL
LIN {X 0,Y 450.08,Z 544.419,A -85,B 0,C 180,E1 -8535.589,E2 -8535.589} C_VEL
LIN {X 0,Y 447.648,Z 544.723,A -85,B 0,C 180,E1 -8536.56,E2 -8536.56} C_VEL
LIN {X 0,Y 446.595,Z 544.854,A -85,B 0,C 180,E1 -8537.31,E2 -8537.31} C_VEL
LIN {X 0,Y 446.507,Z 544.862,A -85,B 0,C 180,E1 -8537.564,E2 -8537.564} C_VEL
LIN {X 0,Y 446.537,Z 544.866,A -85,B 0,C 180,E1 -8540.944,E2 -8540.944} C_VEL
LIN {X 0,Y 446.645,Z 544.845,A -85,B 0,C 180,E1 -8543.676,E2 -8543.676} C_VEL
LIN {X 0,Y 446.707,Z 544.842,A -85,B 0,C 180,E1 -8547.294,E2 -8547.294} C_VEL
LIN {X 0,Y 446.792,Z 544.826,A -85,B 0,C 180,E1 -8549.999,E2 -8549.999} C_VEL
LIN {X 0,Y 446.708,Z 544.838,A -85,B 0,C 180,E1 -8552.705,E2 -8552.705} C_VEL
LIN {X 0,Y 446.637,Z 544.845,A -85,B 0,C 180,E1 -8556.323,E2 -8556.323} C_VEL
LIN {X 0,Y 446.536,Z 544.862,A -85,B 0,C 180,E1 -8559.055,E2 -8559.055} C_VEL
LIN {X 0,Y 446.531,Z 544.859,A -85,B 0,C 180,E1 -8562.729,E2 -8562.729} C_VEL
LIN {X 0,Y 446.487,Z 544.864,A -85,B 0,C 180,E1 -8566.459,E2 -8566.459} C_VEL
LIN {X 0,Y 446.466,Z 544.872,A -85,B 0,C 180,E1 -8569.303,E2 -8569.303} C_VEL
LIN {X 0,Y 446.415,Z 544.874,A -85,B 0,C 180,E1 -8572.199,E2 -8572.199} C_VEL
LIN {X 0,Y 446.454,Z 544.87,A -85,B 0,C 180,E1 -8575.152,E2 -8575.152} C_VEL
LIN {X 0,Y 446.48,Z 544.867,A -85,B 0,C 180,E1 -8578.178,E2 -8578.178} C_VEL
LIN {X 0,Y 446.426,Z 544.874,A -85,B 0,C 180,E1 -8581.299,E2 -8581.299} C_VEL
LIN {X 0,Y 446.426,Z 544.872,A -85,B 0,C 180,E1 -8584.523,E2 -8584.523} C_VEL
LIN {X 0,Y 446.431,Z 544.876,A -85,B 0,C 180,E1 -8588.082,E2 -8588.082} C_VEL
LIN {X 0,Y 446.438,Z 544.87,A -85,B 0,C 180,E1 -8590.92,E2 -8590.92} C_VEL
LIN {X 0,Y 446.412,Z 544.88,A -85,B 0,C 180,E1 -8593.844,E2 -8593.844} C_VEL
LIN {X 0,Y 446.441,Z 544.872,A -85,B 0,C 180,E1 -8596.397,E2 -8596.397} C_VEL
LIN {X 0,Y 446.465,Z 544.871,A -85,B 0,C 180,E1 -8599.805,E2 -8599.805} C_VEL
LIN {X 0,Y 446.43,Z 544.879,A -85,B 0,C 180,E1 -8602.124,E2 -8602.124} C_VEL
LIN {X 0,Y 446.425,Z 544.872,A -85,B 0,C 180,E1 -8605.477,E2 -8605.477} C_VEL
LIN {X 0,Y 446.47,Z 544.984,A -85,B 0,C 180,E1 -8607.171,E2 -8607.171} C_VEL
LIN {X 0,Y 451.774,Z 559.594,A -85,B 0,C 180,E1 -8607.646,E2 -8607.646} C_VEL
LIN {X 0,Y 451.333,Z 604.333,A -85,B 0,C 180,E1 -8608.444,E2 -8608.444} C_VEL
LIN {X 0,Y 451.172,Z 618.121,A -85,B 0,C 180,E1 -8608.865,E2 -8608.865} C_VEL
LIN {X 0,Y 450.878,Z 631.218,A -85,B 0,C 180,E1 -8609.434,E2 -8609.434} C_VEL
LIN {X 0,Y 450.414,Z 644.168,A -85,B 0,C 180,E1 -8610.175,E2 -8610.175} C_VEL
LIN {X 0,Y 449.918,Z 656.036,A -85,B 0,C 180,E1 -8611.038,E2 -8611.038} C_VEL
LIN {X 0,Y 449.284,Z 668.269,A -85,B 0,C 180,E1 -8612.14,E2 -8612.14} C_VEL
LIN {X 0,Y 448.641,Z 679.229,A -85,B 0,C 180,E1 -8613.348,E2 -8613.348} C_VEL
LIN {X 0,Y 448.086,Z 689.273,A -85,B 0,C 180,E1 -8614.698,E2 -8614.698} C_VEL
LIN {X 0,Y 447.533,Z 698.142,A -85,B 0,C 180,E1 -8616.149,E2 -8616.149} C_VEL
LIN {X 0,Y 447.141,Z 705.363,A -85,B 0,C 180,E1 -8617.595,E2 -8617.595} C_VEL
LIN {X 0,Y 446.713,Z 712.083,A -85,B 0,C 180,E1 -8619.269,E2 -8619.269} C_VEL
LIN {X 0,Y 446.488,Z 716.933,A -85,B 0,C 180,E1 -8620.808,E2 -8620.808} C_VEL
LIN {X 0,Y 446.238,Z 721.124,A -85,B 0,C 180,E1 -8622.589,E2 -8622.589} C_VEL
LIN {X 0,Y 446.114,Z 724.048,A -85,B 0,C 180,E1 -8624.466,E2 -8624.466} C_VEL
LIN {X 0,Y 446.103,Z 725.468,A -85,B 0,C 180,E1 -8626.331,E2 -8626.331} C_VEL
LIN {X 0,Y 446.154,Z 725.447,A -85,B 0,C 180,E1 -8628.184,E2 -8628.184} C_VEL
LIN {X 0,Y 446.225,Z 724.052,A -85,B 0,C 180,E1 -8630.024,E2 -8630.024} C_VEL
LIN {X 0,Y 446.403,Z 721.257,A -85,B 0,C 180,E1 -8631.855,E2 -8631.855} C_VEL
LIN {X 0,Y 446.694,Z 718.138,A -85,B 0,C 180,E1 -8633.224,E2 -8633.224} C_VEL
LIN {X 0,Y 446.978,Z 712.676,A -85,B 0,C 180,E1 -8635.039,E2 -8635.039} C_VEL
LIN {X 0,Y 447.376,Z 706.422,A -85,B 0,C 180,E1 -8636.623,E2 -8636.623} C_VEL
LIN {X 0,Y 447.87,Z 698.578,A -85,B 0,C 180,E1 -8638.202,E2 -8638.202} C_VEL
LIN {X 0,Y 448.451,Z 690.337,A -85,B 0,C 180,E1 -8639.551,E2 -8639.551} C_VEL
LIN {X 0,Y 449.057,Z 680.355,A -85,B 0,C 180,E1 -8640.897,E2 -8640.897} C_VEL
LIN {X 0,Y 449.619,Z 670.255,A -85,B 0,C 180,E1 -8642.016,E2 -8642.016} C_VEL
LIN {X 0,Y 450.212,Z 659.21,A -85,B 0,C 180,E1 -8643.02,E2 -8643.02} C_VEL
LIN {X 0,Y 450.765,Z 647.07,A -85,B 0,C 180,E1 -8643.912,E2 -8643.912} C_VEL
LIN {X 0,Y 451.179,Z 633.333,A -85,B 0,C 180,E1 -8644.691,E2 -8644.691} C_VEL
LIN {X 0,Y 451.445,Z 619.33,A -85,B 0,C 180,E1 -8645.276,E2 -8645.276} C_VEL
LIN {X 0,Y 451.477,Z 605.543,A -85,B 0,C 180,E1 -8645.668,E2 -8645.668} C_VEL
LIN {X 0,Y 451.877,Z 559.067,A -85,B 0,C 180,E1 -8646.461,E2 -8646.461} C_VEL
LIN {X 0,Y 446.615,Z 544.856,A -85,B 0,C 180,E1 -8646.977,E2 -8646.977} C_VEL
LIN {X 0,Y 446.524,Z 544.866,A -85,B 0,C 180,E1 -8649.97,E2 -8649.97} C_VEL
LIN {X 0,Y 446.53,Z 544.864,A -85,B 0,C 180,E1 -8652.73,E2 -8652.73} C_VEL
LIN {X 0,Y 446.487,Z 544.868,A -85,B 0,C 180,E1 -8656.46,E2 -8656.46} C_VEL
LIN {X 0,Y 446.466,Z 544.875,A -85,B 0,C 180,E1 -8659.304,E2 -8659.304} C_VEL
LIN {X 0,Y 446.416,Z 544.876,A -85,B 0,C 180,E1 -8662.2,E2 -8662.2} C_VEL
LIN {X 0,Y 446.456,Z 544.874,A -85,B 0,C 180,E1 -8665.153,E2 -8665.153} C_VEL
LIN {X 0,Y 446.482,Z 544.864,A -85,B 0,C 180,E1 -8668.179,E2 -8668.179} C_VEL
LIN {X 0,Y 446.418,Z 544.876,A -85,B 0,C 180,E1 -8671.301,E2 -8671.301} C_VEL
LIN {X 0,Y 446.427,Z 544.868,A -85,B 0,C 180,E1 -8674.524,E2 -8674.524} C_VEL
LIN {X 0,Y 446.428,Z 544.872,A -85,B 0,C 180,E1 -8678.082,E2 -8678.082} C_VEL
LIN {X 0,Y 446.427,Z 544.876,A -85,B 0,C 180,E1 -8680.919,E2 -8680.919} C_VEL
LIN {X 0,Y 446.422,Z 544.874,A -85,B 0,C 180,E1 -8683.844,E2 -8683.844} C_VEL
LIN {X 0,Y 446.398,Z 544.876,A -85,B 0,C 180,E1 -8686.404,E2 -8686.404} C_VEL
LIN {X 0,Y 446.426,Z 544.872,A -85,B 0,C 180,E1 -8689.083,E2 -8689.083} C_VEL
LIN {X 0,Y 446.427,Z 544.876,A -85,B 0,C 180,E1 -8692.124,E2 -8692.124} C_VEL
LIN {X 0,Y 446.482,Z 544.963,A -85,B 0,C 180,E1 -8694.531,E2 -8694.531} C_VEL
LIN {X 0,Y 449.983,Z 561.215,A -85,B 0,C 180,E1 -8697.926,E2 -8697.926} C_VEL
LIN {X 0,Y 450.571,Z 565.423,A -85,B 0,C 180,E1 -8698.76,E2 -8698.76} C_VEL
LIN {X 0,Y 449.479,Z 583.055,A -85,B 0,C 180,E1 -8702.026,E2 -8702.026} C_VEL
LIN {X 0,Y 448.415,Z 603.013,A -85,B 0,C 180,E1 -8705.649,E2 -8705.649} C_VEL
LIN {X 0,Y 447.552,Z 622.202,A -85,B 0,C 180,E1 -8709.069,E2 -8709.069} C_VEL
LIN {X 0,Y 447.015,Z 636.899,A -85,B 0,C 180,E1 -8711.614,E2 -8711.614} C_VEL
LIN {X 0,Y 451.346,Z 670.355,A -85,B 0,C 180,E1 -8712.471,E2 -8712.471} C_VEL
LIN {X 0,Y 449.944,Z 749.52,A -85,B 0,C 180,E1 -8714.021,E2 -8714.021} C_VEL
LIN {X 0,Y 449.345,Z 763.878,A -85,B 0,C 180,E1 -8714.494,E2 -8714.494} C_VEL
LIN {X 0,Y 448.744,Z 776.254,A -85,B 0,C 180,E1 -8715.083,E2 -8715.083} C_VEL
LIN {X 0,Y 448.03,Z 787.899,A -85,B 0,C 180,E1 -8715.813,E2 -8715.813} C_VEL
LIN {X 0,Y 447.492,Z 799.651,A -85,B 0,C 180,E1 -8716.751,E2 -8716.751} C_VEL
LIN {X 0,Y 447.021,Z 809.77,A -85,B 0,C 180,E1 -8717.747,E2 -8717.747} C_VEL
LIN {X 0,Y 446.475,Z 819.231,A -85,B 0,C 180,E1 -8718.883,E2 -8718.883} C_VEL
LIN {X 0,Y 446.09,Z 828.462,A -85,B 0,C 180,E1 -8720.25,E2 -8720.25} C_VEL
LIN {X 0,Y 445.862,Z 835.937,A -85,B 0,C 180,E1 -8721.617,E2 -8721.617} C_VEL
LIN {X 0,Y 445.747,Z 841,A -85,B 0,C 180,E1 -8722.754,E2 -8722.754} C_VEL
LIN {X 0,Y 445.765,Z 845.921,A -85,B 0,C 180,E1 -8724.119,E2 -8724.119} C_VEL
LIN {X 0,Y 445.779,Z 849.673,A -85,B 0,C 180,E1 -8725.479,E2 -8725.479} C_VEL
LIN {X 0,Y 445.804,Z 851.595,A -85,B 0,C 180,E1 -8726.385,E2 -8726.385} C_VEL
LIN {X 0,Y 445.776,Z 853.026,A -85,B 0,C 180,E1 -8727.29,E2 -8727.29} C_VEL
LIN {X 0,Y 445.771,Z 854.006,A -85,B 0,C 180,E1 -8728.194,E2 -8728.194} C_VEL
LIN {X 0,Y 445.769,Z 854.566,A -85,B 0,C 180,E1 -8729.097,E2 -8729.097} C_VEL
LIN {X 0,Y 445.957,Z 854.733,A -85,B 0,C 180,E1 -8730.001,E2 -8730.001} C_VEL
LIN {X 0,Y 445.792,Z 854.393,A -85,B 0,C 180,E1 -8730.904,E2 -8730.904} C_VEL
LIN {X 0,Y 445.817,Z 853.639,A -85,B 0,C 180,E1 -8731.807,E2 -8731.807} C_VEL
LIN {X 0,Y 445.838,Z 852.459,A -85,B 0,C 180,E1 -8732.711,E2 -8732.711} C_VEL
LIN {X 0,Y 445.892,Z 849.84,A -85,B 0,C 180,E1 -8734.068,E2 -8734.068} C_VEL
LIN {X 0,Y 445.837,Z 846.131,A -85,B 0,C 180,E1 -8735.428,E2 -8735.428} C_VEL
LIN {X 0,Y 445.879,Z 841.336,A -85,B 0,C 180,E1 -8736.774,E2 -8736.774} C_VEL
LIN {X 0,Y 445.953,Z 835.126,A -85,B 0,C 180,E1 -8738.155,E2 -8738.155} C_VEL
LIN {X 0,Y 446.069,Z 827.488,A -85,B 0,C 180,E1 -8739.523,E2 -8739.523} C_VEL
LIN {X 0,Y 446.372,Z 818.002,A -85,B 0,C 180,E1 -8740.891,E2 -8740.891} C_VEL
LIN {X 0,Y 446.825,Z 808.37,A -85,B 0,C 180,E1 -8742.029,E2 -8742.029} C_VEL
LIN {X 0,Y 447.141,Z 798.847,A -85,B 0,C 180,E1 -8742.967,E2 -8742.967} C_VEL
LIN {X 0,Y 447.611,Z 787.945,A -85,B 0,C 180,E1 -8743.854,E2 -8743.854} C_VEL
LIN {X 0,Y 448.325,Z 775.88,A -85,B 0,C 180,E1 -8744.642,E2 -8744.642} C_VEL
LIN {X 0,Y 448.95,Z 762.403,A -85,B 0,C 180,E1 -8745.318,E2 -8745.318} C_VEL
LIN {X 0,Y 449.63,Z 748.486,A -85,B 0,C 180,E1 -8745.817,E2 -8745.817} C_VEL
LIN {X 0,Y 449.933,Z 733.788,A -85,B 0,C 180,E1 -8746.155,E2 -8746.155} C_VEL
LIN {X 0,Y 450.736,Z 668.977,A -85,B 0,C 180,E1 -8747.376,E2 -8747.376} C_VEL
LIN {X 0,Y 449.382,Z 654.224,A -85,B 0,C 180,E1 -8747.735,E2 -8747.735} C_VEL
LIN {X 0,Y 447.442,Z 630.351,A -85,B 0,C 180,E1 -8748.328,E2 -8748.328} C_VEL
LIN {X 0,Y 446.758,Z 623.55,A -85,B 0,C 180,E1 -8748.517,E2 -8748.517} C_VEL
LIN {X 0,Y 446.983,Z 604.457,A -85,B 0,C 180,E1 -8751.619,E2 -8751.619} C_VEL
LIN {X 0,Y 447.215,Z 586.071,A -85,B 0,C 180,E1 -8754.65,E2 -8754.65} C_VEL
LIN {X 0,Y 447.475,Z 568.544,A -85,B 0,C 180,E1 -8757.602,E2 -8757.602} C_VEL
LIN {X 0,Y 447.797,Z 553.834,A -85,B 0,C 180,E1 -8760.148,E2 -8760.148} C_VEL
LIN {X 0,Y 447.091,Z 547.796,A -85,B 0,C 180,E1 -8761.248,E2 -8761.248} C_VEL
LIN {X 0,Y 446.535,Z 544.864,A -85,B 0,C 180,E1 -8761.837,E2 -8761.837} C_VEL
LIN {X 0,Y 446.434,Z 544.878,A -85,B 0,C 180,E1 -8765.053,E2 -8765.053} C_VEL
LIN {X 0,Y 446.42,Z 544.874,A -85,B 0,C 180,E1 -8768.079,E2 -8768.079} C_VEL
LIN {X 0,Y 446.432,Z 544.878,A -85,B 0,C 180,E1 -8770.918,E2 -8770.918} C_VEL
LIN {X 0,Y 446.405,Z 544.876,A -85,B 0,C 180,E1 -8773.846,E2 -8773.846} C_VEL
LIN {X 0,Y 446.404,Z 544.878,A -85,B 0,C 180,E1 -8776.403,E2 -8776.403} C_VEL
LIN {X 0,Y 446.432,Z 544.876,A -85,B 0,C 180,E1 -8779.082,E2 -8779.082} C_VEL
LIN {X 0,Y 446.42,Z 544.875,A -85,B 0,C 180,E1 -8781.921,E2 -8781.921} C_VEL
LIN {X 0,Y 446.433,Z 544.874,A -85,B 0,C 180,E1 -8785.477,E2 -8785.477} C_VEL
LIN {X 0,Y 446.421,Z 544.881,A -85,B 0,C 180,E1 -8788.7,E2 -8788.7} C_VEL
LIN {X 0,Y 446.489,Z 544.868,A -85,B 0,C 180,E1 -8791.821,E2 -8791.821} C_VEL
LIN {X 0,Y 446.463,Z 544.876,A -85,B 0,C 180,E1 -8794.848,E2 -8794.848} C_VEL
LIN {X 0,Y 446.453,Z 544.876,A -85,B 0,C 180,E1 -8798.245,E2 -8798.245} C_VEL
LIN {X 0,Y 446.486,Z 544.871,A -85,B 0,C 180,E1 -8800.756,E2 -8800.756} C_VEL
LIN {X 0,Y 448.091,Z 549.215,A -85,B 0,C 180,E1 -8800.922,E2 -8800.922} C_VEL
LIN {X 0,Y 452.63,Z 560.425,A -85,B 0,C 180,E1 -8801.341,E2 -8801.341} C_VEL
LIN {X 0,Y 452.58,Z 593.358,A -85,B 0,C 180,E1 -8801.906,E2 -8801.906} C_VEL
LIN {X 0,Y 452.593,Z 608.04,A -85,B 0,C 180,E1 -8802.333,E2 -8802.333} C_VEL
LIN {X 0,Y 452.378,Z 621.552,A -85,B 0,C 180,E1 -8802.89,E2 -8802.89} C_VEL
LIN {X 0,Y 451.993,Z 635.249,A -85,B 0,C 180,E1 -8803.631,E2 -8803.631} C_VEL
LIN {X 0,Y 451.504,Z 648.446,A -85,B 0,C 180,E1 -8804.54,E2 -8804.54} C_VEL
LIN {X 0,Y 450.918,Z 660.452,A -85,B 0,C 180,E1 -8805.559,E2 -8805.559} C_VEL
LIN {X 0,Y 450.289,Z 671.449,A -85,B 0,C 180,E1 -8806.69,E2 -8806.69} C_VEL
LIN {X 0,Y 449.533,Z 682.434,A -85,B 0,C 180,E1 -8808.044,E2 -8808.044} C_VEL
LIN {X 0,Y 448.839,Z 692.921,A -85,B 0,C 180,E1 -8809.626,E2 -8809.626} C_VEL
LIN {X 0,Y 448.197,Z 701.665,A -85,B 0,C 180,E1 -8811.235,E2 -8811.235} C_VEL
LIN {X 0,Y 447.618,Z 708.617,A -85,B 0,C 180,E1 -8812.784,E2 -8812.784} C_VEL
LIN {X 0,Y 447.299,Z 713.571,A -85,B 0,C 180,E1 -8814.138,E2 -8814.138} C_VEL
LIN {X 0,Y 446.941,Z 718.904,A -85,B 0,C 180,E1 -8815.942,E2 -8815.942} C_VEL
LIN {X 0,Y 446.624,Z 722.045,A -85,B 0,C 180,E1 -8817.294,E2 -8817.294} C_VEL
LIN {X 0,Y 446.407,Z 725.037,A -85,B 0,C 180,E1 -8819.098,E2 -8819.098} C_VEL
LIN {X 0,Y 446.333,Z 726.797,A -85,B 0,C 180,E1 -8820.902,E2 -8820.902} C_VEL
LIN {X 0,Y 446.35,Z 727.379,A -85,B 0,C 180,E1 -8822.707,E2 -8822.707} C_VEL
LIN {X 0,Y 446.226,Z 726.824,A -85,B 0,C 180,E1 -8824.516,E2 -8824.516} C_VEL
LIN {X 0,Y 446.382,Z 725.069,A -85,B 0,C 180,E1 -8826.327,E2 -8826.327} C_VEL
LIN {X 0,Y 446.469,Z 722.12,A -85,B 0,C 180,E1 -8828.144,E2 -8828.144} C_VEL
LIN {X 0,Y 446.668,Z 717.877,A -85,B 0,C 180,E1 -8829.966,E2 -8829.966} C_VEL
LIN {X 0,Y 446.937,Z 712.231,A -85,B 0,C 180,E1 -8831.795,E2 -8831.795} C_VEL
LIN {X 0,Y 447.42,Z 704.99,A -85,B 0,C 180,E1 -8833.628,E2 -8833.628} C_VEL
LIN {X 0,Y 447.935,Z 697.152,A -85,B 0,C 180,E1 -8835.236,E2 -8835.236} C_VEL
LIN {X 0,Y 448.456,Z 688.768,A -85,B 0,C 180,E1 -8836.675,E2 -8836.675} C_VEL
LIN {X 0,Y 449.053,Z 679.618,A -85,B 0,C 180,E1 -8838.005,E2 -8838.005} C_VEL
LIN {X 0,Y 449.772,Z 668.183,A -85,B 0,C 180,E1 -8839.393,E2 -8839.393} C_VEL
LIN {X 0,Y 450.475,Z 656.272,A -85,B 0,C 180,E1 -8840.596,E2 -8840.596} C_VEL
LIN {X 0,Y 451.065,Z 644.403,A -85,B 0,C 180,E1 -8841.598,E2 -8841.598} C_VEL
LIN {X 0,Y 451.647,Z 630.91,A -85,B 0,C 180,E1 -8842.531,E2 -8842.531} C_VEL
LIN {X 0,Y 452.211,Z 616.08,A -85,B 0,C 180,E1 -8843.336,E2 -8843.336} C_VEL
LIN {X 0,Y 452.551,Z 601.276,A -85,B 0,C 180,E1 -8843.944,E2 -8843.944} C_VEL
LIN {X 0,Y 452.694,Z 586.333,A -85,B 0,C 180,E1 -8844.376,E2 -8844.376} C_VEL
LIN {X 0,Y 452.703,Z 561.668,A -85,B 0,C 180,E1 -8844.838,E2 -8844.838} C_VEL
LIN {X 0,Y 446.5,Z 545.093,A -85,B 0,C 180,E1 -8845.399,E2 -8845.399} C_VEL
LIN {X 0,Y 446.466,Z 544.874,A -85,B 0,C 180,E1 -8845.651,E2 -8845.651} C_VEL
LIN {X 0,Y 446.486,Z 544.871,A -85,B 0,C 180,E1 -8848.178,E2 -8848.178} C_VEL
LIN {X 0,Y 446.42,Z 544.876,A -85,B 0,C 180,E1 -8851.774,E2 -8851.774} C_VEL
LIN {X 0,Y 446.43,Z 544.874,A -85,B 0,C 180,E1 -8854.522,E2 -8854.522} C_VEL
LIN {X 0,Y 446.416,Z 544.879,A -85,B 0,C 180,E1 -8858.079,E2 -8858.079} C_VEL
LIN {X 0,Y 446.427,Z 544.872,A -85,B 0,C 180,E1 -8860.917,E2 -8860.917} C_VEL
LIN {X 0,Y 446.4,Z 544.877,A -85,B 0,C 180,E1 -8863.845,E2 -8863.845} C_VEL
LIN {X 0,Y 446.398,Z 544.882,A -85,B 0,C 180,E1 -8866.403,E2 -8866.403} C_VEL
LIN {X 0,Y 446.427,Z 544.872,A -85,B 0,C 180,E1 -8869.082,E2 -8869.082} C_VEL
LIN {X 0,Y 446.43,Z 544.873,A -85,B 0,C 180,E1 -8871.918,E2 -8871.918} C_VEL
LIN {X 0,Y 446.429,Z 544.871,A -85,B 0,C 180,E1 -8875.476,E2 -8875.476} C_VEL
LIN {X 0,Y 446.416,Z 544.879,A -85,B 0,C 180,E1 -8878.699,E2 -8878.699} C_VEL
LIN {X 0,Y 446.484,Z 544.864,A -85,B 0,C 180,E1 -8881.821,E2 -8881.821} C_VEL
LIN {X 0,Y 446.457,Z 544.873,A -85,B 0,C 180,E1 -8884.847,E2 -8884.847} C_VEL
LIN {X 0,Y 446.447,Z 544.871,A -85,B 0,C 180,E1 -8888.244,E2 -8888.244} C_VEL
LIN {X 0,Y 446.456,Z 544.868,A -85,B 0,C 180,E1 -8891.649,E2 -8891.649} C_VEL
LIN {X 0,Y 446.507,Z 544.865,A -85,B 0,C 180,E1 -8894.479,E2 -8894.479} C_VEL
LIN {X 0,Y 446.507,Z 544.862,A -85,B 0,C 180,E1 -8897.564,E2 -8897.564} C_VEL
LIN {X 0,Y 445.828,Z 544.948,A -85,B 0,C 180,E1 -8898.317,E2 -8898.317} C_VEL
LIN {X 0,Y 442.964,Z 545.304,A -85,B 0,C 180,E1 -8899.54,E2 -8899.54} C_VEL
LIN {X 0,Y 440.575,Z 545.603,A -85,B 0,C 180,E1 -8900.526,E2 -8900.526} C_VEL
LIN {X 0,Y 439.588,Z 545.727,A -85,B 0,C 180,E1 -8901.289,E2 -8901.289} C_VEL
LIN {X 0,Y 439.528,Z 545.731,A -85,B 0,C 180,E1 -8901.547,E2 -8901.547} C_VEL
LIN {X 0,Y 439.62,Z 545.721,A -85,B 0,C 180,E1 -8904.495,E2 -8904.495} C_VEL
LIN {X 0,Y 439.634,Z 545.717,A -85,B 0,C 180,E1 -8908.167,E2 -8908.167} C_VEL
LIN {X 0,Y 439.762,Z 545.702,A -85,B 0,C 180,E1 -8909.999,E2 -8909.999} C_VEL
LIN {X 0,Y 439.655,Z 545.717,A -85,B 0,C 180,E1 -8912.748,E2 -8912.748} C_VEL
LIN {X 0,Y 439.609,Z 545.721,A -85,B 0,C 180,E1 -8916.425,E2 -8916.425} C_VEL
LIN {X 0,Y 439.498,Z 545.741,A -85,B 0,C 180,E1 -8919.201,E2 -8919.201} C_VEL
LIN {X 0,Y 439.501,Z 545.735,A -85,B 0,C 180,E1 -8922.726,E2 -8922.726} C_VEL
LIN {X 0,Y 439.444,Z 545.741,A -85,B 0,C 180,E1 -8926.348,E2 -8926.348} C_VEL
LIN {X 0,Y 439.399,Z 545.753,A -85,B 0,C 180,E1 -8929.626,E2 -8929.626} C_VEL
LIN {X 0,Y 439.361,Z 545.751,A -85,B 0,C 180,E1 -8932.575,E2 -8932.575} C_VEL
LIN {X 0,Y 439.402,Z 545.754,A -85,B 0,C 180,E1 -8935.584,E2 -8935.584} C_VEL
LIN {X 0,Y 439.421,Z 545.744,A -85,B 0,C 180,E1 -8938.672,E2 -8938.672} C_VEL
LIN {X 0,Y 439.379,Z 545.753,A -85,B 0,C 180,E1 -8942.033,E2 -8942.033} C_VEL
LIN {X 0,Y 439.391,Z 545.75,A -85,B 0,C 180,E1 -8945.341,E2 -8945.341} C_VEL
LIN {X 0,Y 439.391,Z 545.748,A -85,B 0,C 180,E1 -8948.593,E2 -8948.593} C_VEL
LIN {X 0,Y 439.393,Z 545.748,A -85,B 0,C 180,E1 -8951.258,E2 -8951.258} C_VEL
LIN {X 0,Y 439.399,Z 545.747,A -85,B 0,C 180,E1 -8954.729,E2 -8954.729} C_VEL
LIN {X 0,Y 439.407,Z 545.751,A -85,B 0,C 180,E1 -8957.798,E2 -8957.798} C_VEL
LIN {X 0,Y 439.449,Z 545.746,A -85,B 0,C 180,E1 -8960.23,E2 -8960.23} C_VEL
LIN {X 0,Y 439.372,Z 545.753,A -85,B 0,C 180,E1 -8963.713,E2 -8963.713} C_VEL
